LIN {X 0,Y 258.758,Z 885.566,A -85,B 0,C 180,E1 12350.11,E2 12350.11} C_VEL
LIN {X 0,Y 258.818,Z 883.349,A -85,B 0,C 180,E1 12346.376,E2 12346.376} C_VEL
LIN {X 0,Y 259.397,Z 879.488,A -85,B 0,C 180,E1 12342.915,E2 12342.915} C_VEL
LIN {X 0,Y 260.526,Z 873.775,A -85,B 0,C 180,E1 12339.483,E2 12339.483} C_VEL
LIN {X 0,Y 262.114,Z 866.611,A -85,B 0,C 180,E1 12336.348,E2 12336.348} C_VEL
LIN {X 0,Y 264.269,Z 857.295,A -85,B 0,C 180,E1 12333.25,E2 12333.25} C_VEL
LIN {X 0,Y 266.549,Z 847.181,A -85,B 0,C 180,E1 12330.642,E2 12330.642} C_VEL
LIN {X 0,Y 269.099,Z 835.15,A -85,B 0,C 180,E1 12328.192,E2 12328.192} C_VEL
LIN {X 0,Y 271.468,Z 822.672,A -85,B 0,C 180,E1 12326.196,E2 12326.196} C_VEL
LIN {X 0,Y 273.929,Z 807.744,A -85,B 0,C 180,E1 12324.342,E2 12324.342} C_VEL
LIN {X 0,Y 275.918,Z 792.384,A -85,B 0,C 180,E1 12322.921,E2 12322.921} C_VEL
LIN {X 0,Y 277.442,Z 776.257,A -85,B 0,C 180,E1 12321.847,E2 12321.847} C_VEL
LIN {X 0,Y 278.409,Z 758.677,A -85,B 0,C 180,E1 12321.115,E2 12321.115} C_VEL
LIN {X 0,Y 281.706,Z 674.031,A -85,B 0,C 180,E1 12318.89,E2 12318.89} C_VEL
LIN {X 0,Y 275.076,Z 627.916,A -85,B 0,C 180,E1 12316.6,E2 12316.6} C_VEL
LIN {X 0,Y 278.512,Z 610.893,A -85,B 0,C 180,E1 12313.201,E2 12313.201} C_VEL
LIN {X 0,Y 275.324,Z 596.958,A -85,B 0,C 180,E1 12309.373,E2 12309.373} C_VEL
LIN {X 0,Y 271.574,Z 583.053,A -85,B 0,C 180,E1 12305.183,E2 12305.183} C_VEL
LIN {X 0,Y 267.885,Z 571.432,A -85,B 0,C 180,E1 12301.298,E2 12301.298} C_VEL
LIN {X 0,Y 264.194,Z 560.871,A -85,B 0,C 180,E1 12297.38,E2 12297.38} C_VEL
LIN {X 0,Y 260.854,Z 552.791,A -85,B 0,C 180,E1 12293.977,E2 12293.977} C_VEL
LIN {X 0,Y 259.488,Z 549.45,A -85,B 0,C 180,E1 12292.497,E2 12292.497} C_VEL
LIN {X 0,Y 258.561,Z 546.696,A -85,B 0,C 180,E1 12291.159,E2 12291.159} C_VEL
LIN {X 0,Y 258.551,Z 546.561,A -85,B 0,C 180,E1 12286.317,E2 12286.317} C_VEL
LIN {X 0,Y 258.532,Z 546.552,A -85,B 0,C 180,E1 12281.386,E2 12281.386} C_VEL
LIN {X 0,Y 258.556,Z 546.573,A -85,B 0,C 180,E1 12276.551,E2 12276.551} C_VEL
LIN {X 0,Y 258.554,Z 546.567,A -85,B 0,C 180,E1 12271.708,E2 12271.708} C_VEL
LIN {X 0,Y 258.569,Z 546.551,A -85,B 0,C 180,E1 12267.961,E2 12267.961} C_VEL
LIN {X 0,Y 257.69,Z 546.65,A -85,B 0,C 180,E1 12266.375,E2 12266.375} C_VEL
LIN {X 0,Y 254.009,Z 547.136,A -85,B 0,C 180,E1 12263.744,E2 12263.744} C_VEL
LIN {X 0,Y 250.939,Z 547.534,A -85,B 0,C 180,E1 12261.149,E2 12261.149} C_VEL
LIN {X 0,Y 250.622,Z 547.549,A -85,B 0,C 180,E1 12260.125,E2 12260.125} C_VEL
LIN {X 0,Y 250.618,Z 547.547,A -85,B 0,C 180,E1 12255.107,E2 12255.107} C_VEL
LIN {X 0,Y 250.613,Z 547.525,A -85,B 0,C 180,E1 12250.111,E2 12250.111} C_VEL
LIN {X 0,Y 250.638,Z 547.568,A -85,B 0,C 180,E1 12245.265,E2 12245.265} C_VEL
LIN {X 0,Y 250.61,Z 547.52,A -85,B 0,C 180,E1 12240.229,E2 12240.229} C_VEL
LIN {X 0,Y 250.638,Z 547.563,A -85,B 0,C 180,E1 12235.195,E2 12235.195} C_VEL
LIN {X 0,Y 250.628,Z 547.546,A -85,B 0,C 180,E1 12230.355,E2 12230.355} C_VEL
LIN {X 0,Y 250.629,Z 547.535,A -85,B 0,C 180,E1 12225.208,E2 12225.208} C_VEL
LIN {X 0,Y 250.642,Z 547.549,A -85,B 0,C 180,E1 12220.29,E2 12220.29} C_VEL
LIN {X 0,Y 250.686,Z 547.86,A -85,B 0,C 180,E1 12216.759,E2 12216.759} C_VEL
LIN {X 0,Y 252.116,Z 551.307,A -85,B 0,C 180,E1 12215.142,E2 12215.142} C_VEL
LIN {X 0,Y 254.863,Z 557.484,A -85,B 0,C 180,E1 12212.449,E2 12212.449} C_VEL
LIN {X 0,Y 258.133,Z 564.923,A -85,B 0,C 180,E1 12209.508,E2 12209.508} C_VEL
LIN {X 0,Y 262.832,Z 576.542,A -85,B 0,C 180,E1 12205.471,E2 12205.471} C_VEL
LIN {X 0,Y 267.413,Z 589.235,A -85,B 0,C 180,E1 12201.635,E2 12201.635} C_VEL
LIN {X 0,Y 272.139,Z 603.788,A -85,B 0,C 180,E1 12197.751,E2 12197.751} C_VEL
LIN {X 0,Y 276.856,Z 619.87,A -85,B 0,C 180,E1 12193.999,E2 12193.999} C_VEL
LIN {X 0,Y 277.573,Z 622.236,A -85,B 0,C 180,E1 12193.816,E2 12193.816} C_VEL
LIN {X 0,Y 280.008,Z 658.39,A -85,B 0,C 180,E1 12192.396,E2 12192.396} C_VEL
LIN {X 0,Y 274.15,Z 803.54,A -85,B 0,C 180,E1 12188.817,E2 12188.817} C_VEL
LIN {X 0,Y 272.525,Z 821.816,A -85,B 0,C 180,E1 12188.018,E2 12188.018} C_VEL
LIN {X 0,Y 270.06,Z 839.883,A -85,B 0,C 180,E1 12186.854,E2 12186.854} C_VEL
LIN {X 0,Y 267.199,Z 856.691,A -85,B 0,C 180,E1 12185.367,E2 12185.367} C_VEL
LIN {X 0,Y 263.969,Z 873.171,A -85,B 0,C 180,E1 12183.457,E2 12183.457} C_VEL
LIN {X 0,Y 260.659,Z 888.442,A -85,B 0,C 180,E1 12181.188,E2 12181.188} C_VEL
LIN {X 0,Y 257.395,Z 902.672,A -85,B 0,C 180,E1 12178.542,E2 12178.542} C_VEL
LIN {X 0,Y 254.546,Z 915.418,A -85,B 0,C 180,E1 12175.6,E2 12175.6} C_VEL
LIN {X 0,Y 252.179,Z 926.751,A -85,B 0,C 180,E1 12172.374,E2 12172.374} C_VEL
LIN {X 0,Y 250.447,Z 936.689,A -85,B 0,C 180,E1 12168.868,E2 12168.868} C_VEL
LIN {X 0,Y 249.449,Z 945.396,A -85,B 0,C 180,E1 12164.986,E2 12164.986} C_VEL
LIN {X 0,Y 249.259,Z 952.053,A -85,B 0,C 180,E1 12161.103,E2 12161.103} C_VEL
LIN {X 0,Y 249.653,Z 956.774,A -85,B 0,C 180,E1 12157.365,E2 12157.365} C_VEL
LIN {X 0,Y 250.277,Z 959.854,A -85,B 0,C 180,E1 12153.667,E2 12153.667} C_VEL
LIN {X 0,Y 250.57,Z 961.172,A -85,B 0,C 180,E1 12150.46,E2 12150.46} C_VEL
LIN {X 0,Y 250.268,Z 961.223,A -85,B 0,C 180,E1 12147.175,E2 12147.175} C_VEL
LIN {X 0,Y 249.549,Z 959.846,A -85,B 0,C 180,E1 12143.539,E2 12143.539} C_VEL
LIN {X 0,Y 249.003,Z 956.775,A -85,B 0,C 180,E1 12139.594,E2 12139.594} C_VEL
LIN {X 0,Y 249.15,Z 951.57,A -85,B 0,C 180,E1 12135.273,E2 12135.273} C_VEL
LIN {X 0,Y 250.324,Z 944.676,A -85,B 0,C 180,E1 12131.128,E2 12131.128} C_VEL
LIN {X 0,Y 252.559,Z 936.103,A -85,B 0,C 180,E1 12127.177,E2 12127.177} C_VEL
LIN {X 0,Y 255.721,Z 926.051,A -85,B 0,C 180,E1 12123.535,E2 12123.535} C_VEL
LIN {X 0,Y 259.604,Z 914.488,A -85,B 0,C 180,E1 12120.215,E2 12120.215} C_VEL
LIN {X 0,Y 263.919,Z 901.943,A -85,B 0,C 180,E1 12117.332,E2 12117.332} C_VEL
LIN {X 0,Y 268.723,Z 887.471,A -85,B 0,C 180,E1 12114.688,E2 12114.688} C_VEL
LIN {X 0,Y 273.382,Z 872.233,A -85,B 0,C 180,E1 12112.493,E2 12112.493} C_VEL
LIN {X 0,Y 277.765,Z 856.171,A -85,B 0,C 180,E1 12110.696,E2 12110.696} C_VEL
LIN {X 0,Y 281.501,Z 840.182,A -85,B 0,C 180,E1 12109.332,E2 12109.332} C_VEL
LIN {X 0,Y 284.793,Z 822.514,A -85,B 0,C 180,E1 12108.235,E2 12108.235} C_VEL
LIN {X 0,Y 287.088,Z 804.522,A -85,B 0,C 180,E1 12107.461,E2 12107.461} C_VEL
LIN {X 0,Y 288.669,Z 779.142,A -85,B 0,C 180,E1 12106.785,E2 12106.785} C_VEL
LIN {X 0,Y 295.03,Z 657.964,A -85,B 0,C 180,E1 12103.843,E2 12103.843} C_VEL
LIN {X 0,Y 293.51,Z 637.024,A -85,B 0,C 180,E1 12102.746,E2 12102.746} C_VEL
LIN {X 0,Y 286.069,Z 624.221,A -85,B 0,C 180,E1 12100.516,E2 12100.516} C_VEL
LIN {X 0,Y 284.077,Z 620.553,A -85,B 0,C 180,E1 12099.769,E2 12099.769} C_VEL
LIN {X 0,Y 280.84,Z 610.811,A -85,B 0,C 180,E1 12096.228,E2 12096.228} C_VEL
LIN {X 0,Y 277.656,Z 602.086,A -85,B 0,C 180,E1 12092.449,E2 12092.449} C_VEL
LIN {X 0,Y 274.616,Z 594.628,A -85,B 0,C 180,E1 12088.487,E2 12088.487} C_VEL
LIN {X 0,Y 272.578,Z 590.196,A -85,B 0,C 180,E1 12085.546,E2 12085.546} C_VEL
LIN {X 0,Y 271.016,Z 586.561,A -85,B 0,C 180,E1 12082.791,E2 12082.791} C_VEL
LIN {X 0,Y 269.161,Z 582.502,A -85,B 0,C 180,E1 12078.855,E2 12078.855} C_VEL
LIN {X 0,Y 267.28,Z 578.403,A -85,B 0,C 180,E1 12072.311,E2 12072.311} C_VEL
LIN {X 0,Y 266.55,Z 577.578,A -85,B 0,C 180,E1 12067.11,E2 12067.11} C_VEL
LIN {X 0,Y 266.942,Z 578.179,A -85,B 0,C 180,E1 12062.146,E2 12062.146} C_VEL
LIN {X 0,Y 268.477,Z 582.356,A -85,B 0,C 180,E1 12055.086,E2 12055.086} C_VEL
LIN {X 0,Y 269.944,Z 586.327,A -85,B 0,C 180,E1 12051.05,E2 12051.05} C_VEL
LIN {X 0,Y 271.377,Z 590.311,A -85,B 0,C 180,E1 12047.877,E2 12047.877} C_VEL
LIN {X 0,Y 273.341,Z 595.613,A -85,B 0,C 180,E1 12044.294,E2 12044.294} C_VEL
LIN {X 0,Y 275.612,Z 602.962,A -85,B 0,C 180,E1 12040.282,E2 12040.282} C_VEL
LIN {X 0,Y 277.948,Z 611.166,A -85,B 0,C 180,E1 12036.465,E2 12036.465} C_VEL
LIN {X 0,Y 280.209,Z 620.765,A -85,B 0,C 180,E1 12032.67,E2 12032.67} C_VEL
LIN {X 0,Y 281.533,Z 627.351,A -85,B 0,C 180,E1 12030.418,E2 12030.418} C_VEL
LIN {X 0,Y 283.668,Z 632.135,A -85,B 0,C 180,E1 12029.615,E2 12029.615} C_VEL
LIN {X 0,Y 288.538,Z 660.508,A -85,B 0,C 180,E1 12027.323,E2 12027.323} C_VEL
LIN {X 0,Y 291.484,Z 682.296,A -85,B 0,C 180,E1 12025.844,E2 12025.844} C_VEL
LIN {X 0,Y 286.431,Z 766.945,A -85,B 0,C 180,E1 12023.607,E2 12023.607} C_VEL
LIN {X 0,Y 284.87,Z 783.092,A -85,B 0,C 180,E1 12022.841,E2 12022.841} C_VEL
LIN {X 0,Y 282.515,Z 798.96,A -85,B 0,C 180,E1 12021.731,E2 12021.731} C_VEL
LIN {X 0,Y 279.664,Z 813.068,A -85,B 0,C 180,E1 12020.385,E2 12020.385} C_VEL
LIN {X 0,Y 276.006,Z 827.571,A -85,B 0,C 180,E1 12018.57,E2 12018.57} C_VEL
LIN {X 0,Y 272.149,Z 840.225,A -85,B 0,C 180,E1 12016.51,E2 12016.51} C_VEL
LIN {X 0,Y 268.136,Z 851.743,A -85,B 0,C 180,E1 12014.096,E2 12014.096} C_VEL
LIN {X 0,Y 264.287,Z 861.551,A -85,B 0,C 180,E1 12011.45,E2 12011.45} C_VEL
LIN {X 0,Y 260.567,Z 870.116,A -85,B 0,C 180,E1 12008.428,E2 12008.428} C_VEL
LIN {X 0,Y 257.479,Z 876.685,A -85,B 0,C 180,E1 12005.346,E2 12005.346} C_VEL
LIN {X 0,Y 254.698,Z 882.07,A -85,B 0,C 180,E1 12001.732,E2 12001.732} C_VEL
LIN {X 0,Y 252.737,Z 885.492,A -85,B 0,C 180,E1 11998.079,E2 11998.079} C_VEL
LIN {X 0,Y 251.438,Z 887.087,A -85,B 0,C 180,E1 11994.174,E2 11994.174} C_VEL
LIN {X 0,Y 250.871,Z 886.852,A -85,B 0,C 180,E1 11990.509,E2 11990.509} C_VEL
LIN {X 0,Y 250.867,Z 884.74,A -85,B 0,C 180,E1 11986.672,E2 11986.672} C_VEL
LIN {X 0,Y 251.439,Z 880.947,A -85,B 0,C 180,E1 11983.027,E2 11983.027} C_VEL
LIN {X 0,Y 252.635,Z 875.05,A -85,B 0,C 180,E1 11979.335,E2 11979.335} C_VEL
LIN {X 0,Y 254.287,Z 867.913,A -85,B 0,C 180,E1 11976.091,E2 11976.091} C_VEL
LIN {X 0,Y 256.52,Z 858.641,A -85,B 0,C 180,E1 11972.901,E2 11972.901} C_VEL
LIN {X 0,Y 258.967,Z 848.269,A -85,B 0,C 180,E1 11970.137,E2 11970.137} C_VEL
LIN {X 0,Y 261.661,Z 836.084,A -85,B 0,C 180,E1 11967.589,E2 11967.589} C_VEL
LIN {X 0,Y 264.264,Z 822.893,A -85,B 0,C 180,E1 11965.441,E2 11965.441} C_VEL
LIN {X 0,Y 266.674,Z 808.828,A -85,B 0,C 180,E1 11963.658,E2 11963.658} C_VEL
LIN {X 0,Y 268.614,Z 794.73,A -85,B 0,C 180,E1 11962.297,E2 11962.297} C_VEL
LIN {X 0,Y 270.317,Z 777.953,A -85,B 0,C 180,E1 11961.121,E2 11961.121} C_VEL
LIN {X 0,Y 271.331,Z 761.274,A -85,B 0,C 180,E1 11960.379,E2 11960.379} C_VEL
LIN {X 0,Y 274.846,Z 675.092,A -85,B 0,C 180,E1 11958.055,E2 11958.055} C_VEL
LIN {X 0,Y 268.186,Z 627.499,A -85,B 0,C 180,E1 11955.589,E2 11955.589} C_VEL
LIN {X 0,Y 271.201,Z 613.467,A -85,B 0,C 180,E1 11952.724,E2 11952.724} C_VEL
LIN {X 0,Y 268.053,Z 599.58,A -85,B 0,C 180,E1 11948.787,E2 11948.787} C_VEL
LIN {X 0,Y 264.589,Z 586.434,A -85,B 0,C 180,E1 11944.721,E2 11944.721} C_VEL
LIN {X 0,Y 260.789,Z 574.229,A -85,B 0,C 180,E1 11940.496,E2 11940.496} C_VEL
LIN {X 0,Y 257.249,Z 564.413,A -85,B 0,C 180,E1 11936.684,E2 11936.684} C_VEL
LIN {X 0,Y 253.65,Z 555.043,A -85,B 0,C 180,E1 11932.624,E2 11932.624} C_VEL
LIN {X 0,Y 251.624,Z 550.587,A -85,B 0,C 180,E1 11930.434,E2 11930.434} C_VEL
LIN {X 0,Y 250.629,Z 547.642,A -85,B 0,C 180,E1 11928.834,E2 11928.834} C_VEL
LIN {X 0,Y 250.605,Z 547.576,A -85,B 0,C 180,E1 11923.966,E2 11923.966} C_VEL
LIN {X 0,Y 250.612,Z 547.562,A -85,B 0,C 180,E1 11918.784,E2 11918.784} C_VEL
LIN {X 0,Y 250.614,Z 547.529,A -85,B 0,C 180,E1 11913.92,E2 11913.92} C_VEL
LIN {X 0,Y 250.605,Z 547.561,A -85,B 0,C 180,E1 11908.867,E2 11908.867} C_VEL
LIN {X 0,Y 250.63,Z 547.541,A -85,B 0,C 180,E1 11904.001,E2 11904.001} C_VEL
LIN {X 0,Y 250.622,Z 547.549,A -85,B 0,C 180,E1 11900.125,E2 11900.125} C_VEL
LIN {X 0,Y 249.791,Z 547.637,A -85,B 0,C 180,E1 11898.488,E2 11898.488} C_VEL
LIN {X 0,Y 246.304,Z 548.106,A -85,B 0,C 180,E1 11895.898,E2 11895.898} C_VEL
LIN {X 0,Y 243.012,Z 548.531,A -85,B 0,C 180,E1 11893.093,E2 11893.093} C_VEL
LIN {X 0,Y 242.68,Z 548.551,A -85,B 0,C 180,E1 11892.034,E2 11892.034} C_VEL
LIN {X 0,Y 242.69,Z 548.515,A -85,B 0,C 180,E1 11887.1,E2 11887.1} C_VEL
LIN {X 0,Y 242.673,Z 548.522,A -85,B 0,C 180,E1 11882.126,E2 11882.126} C_VEL
LIN {X 0,Y 242.696,Z 548.552,A -85,B 0,C 180,E1 11877.167,E2 11877.167} C_VEL
LIN {X 0,Y 242.68,Z 548.516,A -85,B 0,C 180,E1 11872.186,E2 11872.186} C_VEL
LIN {X 0,Y 242.695,Z 548.54,A -85,B 0,C 180,E1 11867.146,E2 11867.146} C_VEL
LIN {X 0,Y 242.701,Z 548.561,A -85,B 0,C 180,E1 11862.251,E2 11862.251} C_VEL
LIN {X 0,Y 242.737,Z 548.869,A -85,B 0,C 180,E1 11859.312,E2 11859.312} C_VEL
LIN {X 0,Y 244.971,Z 553.954,A -85,B 0,C 180,E1 11856.678,E2 11856.678} C_VEL
LIN {X 0,Y 247.097,Z 558.693,A -85,B 0,C 180,E1 11854.465,E2 11854.465} C_VEL
LIN {X 0,Y 250.127,Z 565.32,A -85,B 0,C 180,E1 11851.57,E2 11851.57} C_VEL
LIN {X 0,Y 254.559,Z 576.319,A -85,B 0,C 180,E1 11847.445,E2 11847.445} C_VEL
LIN {X 0,Y 259.008,Z 588.256,A -85,B 0,C 180,E1 11843.524,E2 11843.524} C_VEL
LIN {X 0,Y 263.755,Z 602.506,A -85,B 0,C 180,E1 11839.449,E2 11839.449} C_VEL
LIN {X 0,Y 268.597,Z 619.006,A -85,B 0,C 180,E1 11835.287,E2 11835.287} C_VEL
LIN {X 0,Y 269.789,Z 621.934,A -85,B 0,C 180,E1 11834.902,E2 11834.902} C_VEL
LIN {X 0,Y 270.98,Z 624.901,A -85,B 0,C 180,E1 11834.639,E2 11834.639} C_VEL
LIN {X 0,Y 273.194,Z 659.153,A -85,B 0,C 180,E1 11833.257,E2 11833.257} C_VEL
LIN {X 0,Y 267.15,Z 803.024,A -85,B 0,C 180,E1 11829.643,E2 11829.643} C_VEL
LIN {X 0,Y 265.475,Z 821.264,A -85,B 0,C 180,E1 11828.826,E2 11828.826} C_VEL
LIN {X 0,Y 262.989,Z 838.888,A -85,B 0,C 180,E1 11827.67,E2 11827.67} C_VEL
LIN {X 0,Y 260.021,Z 855.79,A -85,B 0,C 180,E1 11826.147,E2 11826.147} C_VEL
LIN {X 0,Y 256.755,Z 871.864,A -85,B 0,C 180,E1 11824.251,E2 11824.251} C_VEL
LIN {X 0,Y 253.317,Z 887.181,A -85,B 0,C 180,E1 11821.932,E2 11821.932} C_VEL
LIN {X 0,Y 249.896,Z 901.455,A -85,B 0,C 180,E1 11819.218,E2 11819.218} C_VEL
LIN {X 0,Y 246.907,Z 914.234,A -85,B 0,C 180,E1 11816.194,E2 11816.194} C_VEL
LIN {X 0,Y 244.415,Z 925.589,A -85,B 0,C 180,E1 11812.87,E2 11812.87} C_VEL
LIN {X 0,Y 242.579,Z 935.542,A -85,B 0,C 180,E1 11809.254,E2 11809.254} C_VEL
LIN {X 0,Y 241.522,Z 944.164,A -85,B 0,C 180,E1 11805.296,E2 11805.296} C_VEL
LIN {X 0,Y 241.3,Z 950.922,A -85,B 0,C 180,E1 11801.232,E2 11801.232} C_VEL
LIN {X 0,Y 241.715,Z 955.639,A -85,B 0,C 180,E1 11797.37,E2 11797.37} C_VEL
LIN {X 0,Y 242.377,Z 958.702,A -85,B 0,C 180,E1 11793.55,E2 11793.55} C_VEL
LIN {X 0,Y 242.665,Z 959.998,A -85,B 0,C 180,E1 11790.239,E2 11790.239} C_VEL
LIN {X 0,Y 242.3,Z 960.012,A -85,B 0,C 180,E1 11786.928,E2 11786.928} C_VEL
LIN {X 0,Y 241.518,Z 958.58,A -85,B 0,C 180,E1 11783.108,E2 11783.108} C_VEL
LIN {X 0,Y 240.994,Z 955.442,A -85,B 0,C 180,E1 11779.002,E2 11779.002} C_VEL
LIN {X 0,Y 241.266,Z 950.307,A -85,B 0,C 180,E1 11774.624,E2 11774.624} C_VEL
LIN {X 0,Y 242.667,Z 943.23,A -85,B 0,C 180,E1 11770.258,E2 11770.258} C_VEL
LIN {X 0,Y 245.175,Z 934.596,A -85,B 0,C 180,E1 11766.193,E2 11766.193} C_VEL
LIN {X 0,Y 248.639,Z 924.487,A -85,B 0,C 180,E1 11762.46,E2 11762.46} C_VEL
LIN {X 0,Y 252.834,Z 912.848,A -85,B 0,C 180,E1 11759.069,E2 11759.069} C_VEL
LIN {X 0,Y 257.636,Z 899.678,A -85,B 0,C 180,E1 11756.03,E2 11756.03} C_VEL
LIN {X 0,Y 262.463,Z 885.824,A -85,B 0,C 180,E1 11753.495,E2 11753.495} C_VEL
LIN {X 0,Y 267.231,Z 870.909,A -85,B 0,C 180,E1 11751.337,E2 11751.337} C_VEL
LIN {X 0,Y 271.819,Z 854.755,A -85,B 0,C 180,E1 11749.524,E2 11749.524} C_VEL
LIN {X 0,Y 275.862,Z 837.898,A -85,B 0,C 180,E1 11748.108,E2 11748.108} C_VEL
LIN {X 0,Y 279.204,Z 820.161,A -85,B 0,C 180,E1 11747.027,E2 11747.027} C_VEL
LIN {X 0,Y 281.553,Z 801.605,A -85,B 0,C 180,E1 11746.251,E2 11746.251} C_VEL
LIN {X 0,Y 283.744,Z 764.34,A -85,B 0,C 180,E1 11745.305,E2 11745.305} C_VEL
LIN {X 0,Y 289.594,Z 658.934,A -85,B 0,C 180,E1 11742.7,E2 11742.7} C_VEL
LIN {X 0,Y 288.373,Z 641.068,A -85,B 0,C 180,E1 11741.736,E2 11741.736} C_VEL
LIN {X 0,Y 280.607,Z 627.479,A -85,B 0,C 180,E1 11739.265,E2 11739.265} C_VEL
LIN {X 0,Y 276.601,Z 620.847,A -85,B 0,C 180,E1 11737.753,E2 11737.753} C_VEL
LIN {X 0,Y 273.257,Z 611.063,A -85,B 0,C 180,E1 11733.791,E2 11733.791} C_VEL
LIN {X 0,Y 270.295,Z 603.354,A -85,B 0,C 180,E1 11729.959,E2 11729.959} C_VEL
LIN {X 0,Y 267.793,Z 597.058,A -85,B 0,C 180,E1 11726.14,E2 11726.14} C_VEL
LIN {X 0,Y 265.692,Z 592.469,A -85,B 0,C 180,E1 11722.572,E2 11722.572} C_VEL
LIN {X 0,Y 264.006,Z 588.611,A -85,B 0,C 180,E1 11718.779,E2 11718.779} C_VEL
LIN {X 0,Y 262.172,Z 584.562,A -85,B 0,C 180,E1 11712.331,E2 11712.331} C_VEL
LIN {X 0,Y 261.41,Z 583.713,A -85,B 0,C 180,E1 11707.03,E2 11707.03} C_VEL
LIN {X 0,Y 261.77,Z 584.358,A -85,B 0,C 180,E1 11701.97,E2 11701.97} C_VEL
LIN {X 0,Y 263.12,Z 588.296,A -85,B 0,C 180,E1 11695.204,E2 11695.204} C_VEL
LIN {X 0,Y 264.525,Z 592.307,A -85,B 0,C 180,E1 11691.084,E2 11691.084} C_VEL
LIN {X 0,Y 265.874,Z 596.287,A -85,B 0,C 180,E1 11687.842,E2 11687.842} C_VEL
LIN {X 0,Y 267.657,Z 601.313,A -85,B 0,C 180,E1 11684.397,E2 11684.397} C_VEL
LIN {X 0,Y 269.971,Z 609.092,A -85,B 0,C 180,E1 11680.078,E2 11680.078} C_VEL
LIN {X 0,Y 272.166,Z 617.547,A -85,B 0,C 180,E1 11676.153,E2 11676.153} C_VEL
LIN {X 0,Y 274.175,Z 626.767,A -85,B 0,C 180,E1 11672.527,E2 11672.527} C_VEL
LIN {X 0,Y 278.927,Z 636.071,A -85,B 0,C 180,E1 11670.675,E2 11670.675} C_VEL
LIN {X 0,Y 283.381,Z 663.273,A -85,B 0,C 180,E1 11668.416,E2 11668.416} C_VEL
LIN {X 0,Y 286.018,Z 683.721,A -85,B 0,C 180,E1 11666.987,E2 11666.987} C_VEL
LIN {X 0,Y 280.793,Z 767.637,A -85,B 0,C 180,E1 11664.746,E2 11664.746} C_VEL
LIN {X 0,Y 279.152,Z 783.83,A -85,B 0,C 180,E1 11663.969,E2 11663.969} C_VEL
LIN {X 0,Y 276.671,Z 799.801,A -85,B 0,C 180,E1 11662.838,E2 11662.838} C_VEL
LIN {X 0,Y 273.599,Z 814.23,A -85,B 0,C 180,E1 11661.439,E2 11661.439} C_VEL
LIN {X 0,Y 269.746,Z 828.724,A -85,B 0,C 180,E1 11659.59,E2 11659.59} C_VEL
LIN {X 0,Y 265.72,Z 841.244,A -85,B 0,C 180,E1 11657.511,E2 11657.511} C_VEL
LIN {X 0,Y 261.301,Z 853.247,A -85,B 0,C 180,E1 11654.935,E2 11654.935} C_VEL
LIN {X 0,Y 257.266,Z 862.926,A -85,B 0,C 180,E1 11652.241,E2 11652.241} C_VEL
LIN {X 0,Y 253.347,Z 871.438,A -85,B 0,C 180,E1 11649.15,E2 11649.15} C_VEL
LIN {X 0,Y 250.075,Z 877.958,A -85,B 0,C 180,E1 11645.99,E2 11645.99} C_VEL
LIN {X 0,Y 247.096,Z 883.341,A -85,B 0,C 180,E1 11642.251,E2 11642.251} C_VEL
LIN {X 0,Y 245.006,Z 886.709,A -85,B 0,C 180,E1 11638.514,E2 11638.514} C_VEL
LIN {X 0,Y 243.597,Z 888.292,A -85,B 0,C 180,E1 11634.486,E2 11634.486} C_VEL
LIN {X 0,Y 242.971,Z 888.056,A -85,B 0,C 180,E1 11630.721,E2 11630.721} C_VEL
LIN {X 0,Y 242.938,Z 885.938,A -85,B 0,C 180,E1 11626.74,E2 11626.74} C_VEL
LIN {X 0,Y 243.5,Z 882.258,A -85,B 0,C 180,E1 11623.048,E2 11623.048} C_VEL
LIN {X 0,Y 244.651,Z 876.713,A -85,B 0,C 180,E1 11619.405,E2 11619.405} C_VEL
LIN {X 0,Y 246.333,Z 869.723,A -85,B 0,C 180,E1 11616.034,E2 11616.034} C_VEL
LIN {X 0,Y 248.591,Z 860.689,A -85,B 0,C 180,E1 11612.763,E2 11612.763} C_VEL
LIN {X 0,Y 251.015,Z 850.942,A -85,B 0,C 180,E1 11609.997,E2 11609.997} C_VEL
LIN {X 0,Y 253.732,Z 839.277,A -85,B 0,C 180,E1 11607.4,E2 11607.4} C_VEL
LIN {X 0,Y 256.535,Z 826.024,A -85,B 0,C 180,E1 11605.079,E2 11605.079} C_VEL
LIN {X 0,Y 259.178,Z 811.47,A -85,B 0,C 180,E1 11603.129,E2 11603.129} C_VEL
LIN {X 0,Y 261.336,Z 796.944,A -85,B 0,C 180,E1 11601.638,E2 11601.638} C_VEL
LIN {X 0,Y 263.132,Z 780.437,A -85,B 0,C 180,E1 11600.421,E2 11600.421} C_VEL
LIN {X 0,Y 264.262,Z 764.216,A -85,B 0,C 180,E1 11599.628,E2 11599.628} C_VEL
LIN {X 0,Y 267.998,Z 676.088,A -85,B 0,C 180,E1 11597.186,E2 11597.186} C_VEL
LIN {X 0,Y 261.343,Z 627.714,A -85,B 0,C 180,E1 11594.606,E2 11594.606} C_VEL
LIN {X 0,Y 263.831,Z 615.702,A -85,B 0,C 180,E1 11592.122,E2 11592.122} C_VEL
LIN {X 0,Y 260.776,Z 601.953,A -85,B 0,C 180,E1 11588.106,E2 11588.106} C_VEL
LIN {X 0,Y 257.4,Z 589.044,A -85,B 0,C 180,E1 11583.963,E2 11583.963} C_VEL
LIN {X 0,Y 253.675,Z 577.144,A -85,B 0,C 180,E1 11579.677,E2 11579.677} C_VEL
LIN {X 0,Y 250.192,Z 567.11,A -85,B 0,C 180,E1 11575.635,E2 11575.635} C_VEL
LIN {X 0,Y 246.799,Z 558.83,A -85,B 0,C 180,E1 11571.81,E2 11571.81} C_VEL
LIN {X 0,Y 245.287,Z 555.284,A -85,B 0,C 180,E1 11570.027,E2 11570.027} C_VEL
LIN {X 0,Y 243.895,Z 551.902,A -85,B 0,C 180,E1 11568.256,E2 11568.256} C_VEL
LIN {X 0,Y 242.694,Z 548.684,A -85,B 0,C 180,E1 11566.381,E2 11566.381} C_VEL
LIN {X 0,Y 242.655,Z 548.527,A -85,B 0,C 180,E1 11561.246,E2 11561.246} C_VEL
LIN {X 0,Y 242.682,Z 548.543,A -85,B 0,C 180,E1 11556.391,E2 11556.391} C_VEL
LIN {X 0,Y 242.667,Z 548.552,A -85,B 0,C 180,E1 11551.276,E2 11551.276} C_VEL
LIN {X 0,Y 242.683,Z 548.509,A -85,B 0,C 180,E1 11546.158,E2 11546.158} C_VEL
LIN {X 0,Y 242.679,Z 548.564,A -85,B 0,C 180,E1 11541.259,E2 11541.259} C_VEL
LIN {X 0,Y 242.68,Z 548.516,A -85,B 0,C 180,E1 11536.025,E2 11536.025} C_VEL
LIN {X 0,Y 242.68,Z 548.551,A -85,B 0,C 180,E1 11532.034,E2 11532.034} C_VEL
LIN {X 0,Y 241.836,Z 548.633,A -85,B 0,C 180,E1 11530.344,E2 11530.344} C_VEL
LIN {X 0,Y 238.349,Z 549.094,A -85,B 0,C 180,E1 11527.667,E2 11527.667} C_VEL
LIN {X 0,Y 235.072,Z 549.519,A -85,B 0,C 180,E1 11524.766,E2 11524.766} C_VEL
LIN {X 0,Y 234.747,Z 549.542,A -85,B 0,C 180,E1 11523.672,E2 11523.672} C_VEL
LIN {X 0,Y 234.751,Z 549.505,A -85,B 0,C 180,E1 11518.78,E2 11518.78} C_VEL
LIN {X 0,Y 234.742,Z 549.511,A -85,B 0,C 180,E1 11513.642,E2 11513.642} C_VEL
LIN {X 0,Y 234.765,Z 549.556,A -85,B 0,C 180,E1 11508.702,E2 11508.702} C_VEL
LIN {X 0,Y 234.748,Z 549.525,A -85,B 0,C 180,E1 11503.397,E2 11503.397} C_VEL
LIN {X 0,Y 234.813,Z 549.902,A -85,B 0,C 180,E1 11502.211,E2 11502.211} C_VEL
LIN {X 0,Y 236.511,Z 553.639,A -85,B 0,C 180,E1 11499.975,E2 11499.975} C_VEL
LIN {X 0,Y 239.177,Z 559.522,A -85,B 0,C 180,E1 11496.862,E2 11496.862} C_VEL
LIN {X 0,Y 242.464,Z 566.618,A -85,B 0,C 180,E1 11493.486,E2 11493.486} C_VEL
LIN {X 0,Y 246.915,Z 577.538,A -85,B 0,C 180,E1 11489.051,E2 11489.051} C_VEL
LIN {X 0,Y 251.237,Z 588.998,A -85,B 0,C 180,E1 11485.035,E2 11485.035} C_VEL
LIN {X 0,Y 255.941,Z 603.128,A -85,B 0,C 180,E1 11480.738,E2 11480.738} C_VEL
LIN {X 0,Y 260.38,Z 618.15,A -85,B 0,C 180,E1 11476.73,E2 11476.73} C_VEL
LIN {X 0,Y 261.29,Z 620.86,A -85,B 0,C 180,E1 11476.201,E2 11476.201} C_VEL
LIN {X 0,Y 264.444,Z 627.738,A -85,B 0,C 180,E1 11475.492,E2 11475.492} C_VEL
LIN {X 0,Y 266.429,Z 659.847,A -85,B 0,C 180,E1 11474.159,E2 11474.159} C_VEL
LIN {X 0,Y 260.175,Z 802.403,A -85,B 0,C 180,E1 11470.501,E2 11470.501} C_VEL
LIN {X 0,Y 258.451,Z 820.641,A -85,B 0,C 180,E1 11469.667,E2 11469.667} C_VEL
LIN {X 0,Y 255.879,Z 838.284,A -85,B 0,C 180,E1 11468.485,E2 11468.485} C_VEL
LIN {X 0,Y 252.847,Z 855.007,A -85,B 0,C 180,E1 11466.946,E2 11466.946} C_VEL
LIN {X 0,Y 249.413,Z 871.298,A -85,B 0,C 180,E1 11464.978,E2 11464.978} C_VEL
LIN {X 0,Y 245.858,Z 886.538,A -85,B 0,C 180,E1 11462.606,E2 11462.606} C_VEL
LIN {X 0,Y 242.292,Z 900.804,A -85,B 0,C 180,E1 11459.812,E2 11459.812} C_VEL
LIN {X 0,Y 239.082,Z 913.947,A -85,B 0,C 180,E1 11456.583,E2 11456.583} C_VEL
LIN {X 0,Y 236.51,Z 925.175,A -85,B 0,C 180,E1 11453.152,E2 11453.152} C_VEL
LIN {X 0,Y 234.623,Z 935.007,A -85,B 0,C 180,E1 11449.416,E2 11449.416} C_VEL
LIN {X 0,Y 233.562,Z 943.343,A -85,B 0,C 180,E1 11445.393,E2 11445.393} C_VEL
LIN {X 0,Y 233.354,Z 950.116,A -85,B 0,C 180,E1 11441.119,E2 11441.119} C_VEL
LIN {X 0,Y 233.817,Z 954.722,A -85,B 0,C 180,E1 11437.126,E2 11437.126} C_VEL
LIN {X 0,Y 234.518,Z 957.664,A -85,B 0,C 180,E1 11433.18,E2 11433.18} C_VEL
LIN {X 0,Y 234.745,Z 958.874,A -85,B 0,C 180,E1 11429.759,E2 11429.759} C_VEL
LIN {X 0,Y 234.258,Z 958.735,A -85,B 0,C 180,E1 11426.333,E2 11426.333} C_VEL
LIN {X 0,Y 233.392,Z 957.002,A -85,B 0,C 180,E1 11422.124,E2 11422.124} C_VEL
LIN {X 0,Y 232.991,Z 953.372,A -85,B 0,C 180,E1 11417.614,E2 11417.614} C_VEL
LIN {X 0,Y 233.612,Z 947.891,A -85,B 0,C 180,E1 11413.084,E2 11413.084} C_VEL
LIN {X 0,Y 235.47,Z 940.434,A -85,B 0,C 180,E1 11408.587,E2 11408.587} C_VEL
LIN {X 0,Y 238.497,Z 931.353,A -85,B 0,C 180,E1 11404.423,E2 11404.423} C_VEL
LIN {X 0,Y 242.479,Z 920.741,A -85,B 0,C 180,E1 11400.62,E2 11400.62} C_VEL
LIN {X 0,Y 247.197,Z 908.587,A -85,B 0,C 180,E1 11397.187,E2 11397.187} C_VEL
LIN {X 0,Y 252.318,Z 895.326,A -85,B 0,C 180,E1 11394.24,E2 11394.24} C_VEL
LIN {X 0,Y 257.445,Z 880.96,A -85,B 0,C 180,E1 11391.731,E2 11391.731} C_VEL
LIN {X 0,Y 262.426,Z 865.653,A -85,B 0,C 180,E1 11389.639,E2 11389.639} C_VEL
LIN {X 0,Y 267.068,Z 849.369,A -85,B 0,C 180,E1 11387.93,E2 11387.93} C_VEL
LIN {X 0,Y 271.101,Z 832.39,A -85,B 0,C 180,E1 11386.599,E2 11386.599} C_VEL
LIN {X 0,Y 274.344,Z 814.44,A -85,B 0,C 180,E1 11385.592,E2 11385.592} C_VEL
LIN {X 0,Y 276.379,Z 796.193,A -85,B 0,C 180,E1 11384.914,E2 11384.914} C_VEL
LIN {X 0,Y 284.285,Z 660.052,A -85,B 0,C 180,E1 11381.52,E2 11381.52} C_VEL
LIN {X 0,Y 283.321,Z 645.072,A -85,B 0,C 180,E1 11380.685,E2 11380.685} C_VEL
LIN {X 0,Y 276.399,Z 632.744,A -85,B 0,C 180,E1 11378.344,E2 11378.344} C_VEL
LIN {X 0,Y 269.173,Z 621.266,A -85,B 0,C 180,E1 11375.544,E2 11375.544} C_VEL
LIN {X 0,Y 266.214,Z 612.784,A -85,B 0,C 180,E1 11371.723,E2 11371.723} C_VEL
LIN {X 0,Y 263.514,Z 605.816,A -85,B 0,C 180,E1 11367.82,E2 11367.82} C_VEL
LIN {X 0,Y 261.513,Z 601.238,A -85,B 0,C 180,E1 11364.629,E2 11364.629} C_VEL
LIN {X 0,Y 260.378,Z 598.381,A -85,B 0,C 180,E1 11362.343,E2 11362.343} C_VEL
LIN {X 0,Y 258.835,Z 594.706,A -85,B 0,C 180,E1 11358.7,E2 11358.7} C_VEL
LIN {X 0,Y 257.012,Z 590.659,A -85,B 0,C 180,E1 11352.126,E2 11352.126} C_VEL
LIN {X 0,Y 256.291,Z 589.864,A -85,B 0,C 180,E1 11346.946,E2 11346.946} C_VEL
LIN {X 0,Y 256.608,Z 590.483,A -85,B 0,C 180,E1 11342.009,E2 11342.009} C_VEL
LIN {X 0,Y 257.808,Z 594.323,A -85,B 0,C 180,E1 11335.269,E2 11335.269} C_VEL
LIN {X 0,Y 259.03,Z 598.001,A -85,B 0,C 180,E1 11331.341,E2 11331.341} C_VEL
LIN {X 0,Y 260.3,Z 601.971,A -85,B 0,C 180,E1 11328.028,E2 11328.028} C_VEL
LIN {X 0,Y 261.963,Z 607.026,A -85,B 0,C 180,E1 11324.503,E2 11324.503} C_VEL
LIN {X 0,Y 264.07,Z 614.397,A -85,B 0,C 180,E1 11320.306,E2 11320.306} C_VEL
LIN {X 0,Y 266.141,Z 622.874,A -85,B 0,C 180,E1 11316.297,E2 11316.297} C_VEL
LIN {X 0,Y 267.043,Z 626.745,A -85,B 0,C 180,E1 11314.732,E2 11314.732} C_VEL
LIN {X 0,Y 273.518,Z 638.658,A -85,B 0,C 180,E1 11312.071,E2 11312.071} C_VEL
LIN {X 0,Y 274.606,Z 641.493,A -85,B 0,C 180,E1 11311.63,E2 11311.63} C_VEL
LIN {X 0,Y 278.917,Z 670.354,A -85,B 0,C 180,E1 11309.22,E2 11309.22} C_VEL
LIN {X 0,Y 280.644,Z 685.535,A -85,B 0,C 180,E1 11308.164,E2 11308.164} C_VEL
LIN {X 0,Y 275.263,Z 768.44,A -85,B 0,C 180,E1 11305.926,E2 11305.926} C_VEL
LIN {X 0,Y 273.516,Z 784.785,A -85,B 0,C 180,E1 11305.129,E2 11305.129} C_VEL
LIN {X 0,Y 270.955,Z 800.527,A -85,B 0,C 180,E1 11304.002,E2 11304.002} C_VEL
LIN {X 0,Y 267.633,Z 815.416,A -85,B 0,C 180,E1 11302.539,E2 11302.539} C_VEL
LIN {X 0,Y 263.627,Z 829.776,A -85,B 0,C 180,E1 11300.678,E2 11300.678} C_VEL
LIN {X 0,Y 259.439,Z 842.188,A -85,B 0,C 180,E1 11298.586,E2 11298.586} C_VEL
LIN {X 0,Y 254.868,Z 853.983,A -85,B 0,C 180,E1 11296.021,E2 11296.021} C_VEL
LIN {X 0,Y 250.652,Z 863.613,A -85,B 0,C 180,E1 11293.315,E2 11293.315} C_VEL
LIN {X 0,Y 246.465,Z 872.186,A -85,B 0,C 180,E1 11290.16,E2 11290.16} C_VEL
LIN {X 0,Y 242.706,Z 879.228,A -85,B 0,C 180,E1 11286.673,E2 11286.673} C_VEL
LIN {X 0,Y 239.552,Z 884.553,A -85,B 0,C 180,E1 11282.854,E2 11282.854} C_VEL
LIN {X 0,Y 237.292,Z 887.927,A -85,B 0,C 180,E1 11278.978,E2 11278.978} C_VEL
LIN {X 0,Y 235.764,Z 889.496,A -85,B 0,C 180,E1 11274.82,E2 11274.82} C_VEL
LIN {X 0,Y 235.071,Z 889.254,A -85,B 0,C 180,E1 11270.929,E2 11270.929} C_VEL
LIN {X 0,Y 235.008,Z 887.13,A -85,B 0,C 180,E1 11266.806,E2 11266.806} C_VEL
LIN {X 0,Y 235.576,Z 883.463,A -85,B 0,C 180,E1 11262.996,E2 11262.996} C_VEL
LIN {X 0,Y 236.763,Z 877.935,A -85,B 0,C 180,E1 11259.231,E2 11259.231} C_VEL
LIN {X 0,Y 238.491,Z 871.016,A -85,B 0,C 180,E1 11255.771,E2 11255.771} C_VEL
LIN {X 0,Y 240.662,Z 862.714,A -85,B 0,C 180,E1 11252.616,E2 11252.616} C_VEL
LIN {X 0,Y 243.367,Z 852.284,A -85,B 0,C 180,E1 11249.526,E2 11249.526} C_VEL
LIN {X 0,Y 246.191,Z 840.726,A -85,B 0,C 180,E1 11246.854,E2 11246.854} C_VEL
LIN {X 0,Y 249.142,Z 827.372,A -85,B 0,C 180,E1 11244.436,E2 11244.436} C_VEL
LIN {X 0,Y 251.844,Z 813.244,A -85,B 0,C 180,E1 11242.47,E2 11242.47} C_VEL
LIN {X 0,Y 254.249,Z 797.828,A -85,B 0,C 180,E1 11240.834,E2 11240.834} C_VEL
LIN {X 0,Y 256.123,Z 781.395,A -85,B 0,C 180,E1 11239.589,E2 11239.589} C_VEL
LIN {X 0,Y 257.33,Z 764.93,A -85,B 0,C 180,E1 11238.76,E2 11238.76} C_VEL
LIN {X 0,Y 261.224,Z 677.185,A -85,B 0,C 180,E1 11236.279,E2 11236.279} C_VEL
LIN {X 0,Y 254.565,Z 627.292,A -85,B 0,C 180,E1 11233.513,E2 11233.513} C_VEL
LIN {X 0,Y 256.559,Z 618.329,A -85,B 0,C 180,E1 11231.597,E2 11231.597} C_VEL
LIN {X 0,Y 253.497,Z 604.271,A -85,B 0,C 180,E1 11227.364,E2 11227.364} C_VEL
LIN {X 0,Y 250.209,Z 591.672,A -85,B 0,C 180,E1 11223.156,E2 11223.156} C_VEL
LIN {X 0,Y 246.573,Z 579.842,A -85,B 0,C 180,E1 11218.732,E2 11218.732} C_VEL
LIN {X 0,Y 243.308,Z 570.733,A -85,B 0,C 180,E1 11214.864,E2 11214.864} C_VEL
LIN {X 0,Y 240.456,Z 563.47,A -85,B 0,C 180,E1 11211.411,E2 11211.411} C_VEL
LIN {X 0,Y 238.165,Z 557.559,A -85,B 0,C 180,E1 11208.356,E2 11208.356} C_VEL
LIN {X 0,Y 236.025,Z 553.02,A -85,B 0,C 180,E1 11205.655,E2 11205.655} C_VEL
LIN {X 0,Y 234.734,Z 549.649,A -85,B 0,C 180,E1 11203.446,E2 11203.446} C_VEL
LIN {X 0,Y 234.75,Z 549.543,A -85,B 0,C 180,E1 11198.401,E2 11198.401} C_VEL
LIN {X 0,Y 234.721,Z 549.508,A -85,B 0,C 180,E1 11193.334,E2 11193.334} C_VEL
LIN {X 0,Y 234.752,Z 549.515,A -85,B 0,C 180,E1 11188.16,E2 11188.16} C_VEL
LIN {X 0,Y 234.731,Z 549.538,A -85,B 0,C 180,E1 11183.067,E2 11183.067} C_VEL
LIN {X 0,Y 234.747,Z 549.492,A -85,B 0,C 180,E1 11177.859,E2 11177.859} C_VEL
LIN {X 0,Y 234.737,Z 549.555,A -85,B 0,C 180,E1 11172.738,E2 11172.738} C_VEL
LIN {X 0,Y 234.754,Z 549.496,A -85,B 0,C 180,E1 11167.588,E2 11167.588} C_VEL
LIN {X 0,Y 234.747,Z 549.542,A -85,B 0,C 180,E1 11163.672,E2 11163.672} C_VEL
LIN {X 0,Y 233.918,Z 549.624,A -85,B 0,C 180,E1 11161.924,E2 11161.924} C_VEL
LIN {X 0,Y 230.455,Z 550.075,A -85,B 0,C 180,E1 11159.155,E2 11159.155} C_VEL
LIN {X 0,Y 227.166,Z 550.502,A -85,B 0,C 180,E1 11156.153,E2 11156.153} C_VEL
LIN {X 0,Y 226.82,Z 550.519,A -85,B 0,C 180,E1 11155.02,E2 11155.02} C_VEL
LIN {X 0,Y 226.804,Z 550.519,A -85,B 0,C 180,E1 11149.844,E2 11149.844} C_VEL
LIN {X 0,Y 226.846,Z 550.795,A -85,B 0,C 180,E1 11145.711,E2 11145.711} C_VEL
LIN {X 0,Y 228.651,Z 554.73,A -85,B 0,C 180,E1 11142.964,E2 11142.964} C_VEL
LIN {X 0,Y 231.527,Z 560.935,A -85,B 0,C 180,E1 11139.261,E2 11139.261} C_VEL
LIN {X 0,Y 233.574,Z 565.551,A -85,B 0,C 180,E1 11136.808,E2 11136.808} C_VEL
LIN {X 0,Y 236.356,Z 571.494,A -85,B 0,C 180,E1 11133.9,E2 11133.9} C_VEL
LIN {X 0,Y 240.54,Z 581.95,A -85,B 0,C 180,E1 11129.528,E2 11129.528} C_VEL
LIN {X 0,Y 244.763,Z 593.431,A -85,B 0,C 180,E1 11125.402,E2 11125.402} C_VEL
LIN {X 0,Y 249.37,Z 607.597,A -85,B 0,C 180,E1 11120.987,E2 11120.987} C_VEL
LIN {X 0,Y 253.183,Z 620.447,A -85,B 0,C 180,E1 11117.522,E2 11117.522} C_VEL
LIN {X 0,Y 257.966,Z 630.596,A -85,B 0,C 180,E1 11116.387,E2 11116.387} C_VEL
LIN {X 0,Y 259.728,Z 660.675,A -85,B 0,C 180,E1 11115.103,E2 11115.103} C_VEL
LIN {X 0,Y 253.27,Z 801.678,A -85,B 0,C 180,E1 11111.41,E2 11111.41} C_VEL
LIN {X 0,Y 251.493,Z 819.934,A -85,B 0,C 180,E1 11110.558,E2 11110.558} C_VEL
LIN {X 0,Y 248.81,Z 837.73,A -85,B 0,C 180,E1 11109.34,E2 11109.34} C_VEL
LIN {X 0,Y 245.641,Z 854.579,A -85,B 0,C 180,E1 11107.749,E2 11107.749} C_VEL
LIN {X 0,Y 242.123,Z 870.608,A -85,B 0,C 180,E1 11105.756,E2 11105.756} C_VEL
LIN {X 0,Y 238.433,Z 885.806,A -85,B 0,C 180,E1 11103.322,E2 11103.322} C_VEL
LIN {X 0,Y 234.734,Z 900.011,A -85,B 0,C 180,E1 11100.457,E2 11100.457} C_VEL
LIN {X 0,Y 231.491,Z 912.722,A -85,B 0,C 180,E1 11097.248,E2 11097.248} C_VEL
LIN {X 0,Y 228.777,Z 924.001,A -85,B 0,C 180,E1 11093.71,E2 11093.71} C_VEL
LIN {X 0,Y 226.77,Z 933.86,A -85,B 0,C 180,E1 11089.848,E2 11089.848} C_VEL
LIN {X 0,Y 225.631,Z 942.204,A -85,B 0,C 180,E1 11085.685,E2 11085.685} C_VEL
LIN {X 0,Y 225.395,Z 948.977,A -85,B 0,C 180,E1 11081.258,E2 11081.258} C_VEL
LIN {X 0,Y 225.924,Z 953.804,A -85,B 0,C 180,E1 11076.865,E2 11076.865} C_VEL
LIN {X 0,Y 226.622,Z 956.505,A -85,B 0,C 180,E1 11073.038,E2 11073.038} C_VEL
LIN {X 0,Y 226.84,Z 957.634,A -85,B 0,C 180,E1 11069.751,E2 11069.751} C_VEL
LIN {X 0,Y 226.3,Z 957.55,A -85,B 0,C 180,E1 11066.203,E2 11066.203} C_VEL
LIN {X 0,Y 225.391,Z 955.861,A -85,B 0,C 180,E1 11061.843,E2 11061.843} C_VEL
LIN {X 0,Y 225.026,Z 952.279,A -85,B 0,C 180,E1 11057.168,E2 11057.168} C_VEL
LIN {X 0,Y 225.772,Z 946.864,A -85,B 0,C 180,E1 11052.478,E2 11052.478} C_VEL
LIN {X 0,Y 227.83,Z 939.493,A -85,B 0,C 180,E1 11047.831,E2 11047.831} C_VEL
LIN {X 0,Y 231.106,Z 930.472,A -85,B 0,C 180,E1 11043.543,E2 11043.543} C_VEL
LIN {X 0,Y 235.357,Z 919.914,A -85,B 0,C 180,E1 11039.639,E2 11039.639} C_VEL
LIN {X 0,Y 240.363,Z 907.819,A -85,B 0,C 180,E1 11036.13,E2 11036.13} C_VEL
LIN {X 0,Y 245.753,Z 894.666,A -85,B 0,C 180,E1 11033.129,E2 11033.129} C_VEL
LIN {X 0,Y 251.22,Z 880.193,A -85,B 0,C 180,E1 11030.544,E2 11030.544} C_VEL
LIN {X 0,Y 256.327,Z 865.252,A -85,B 0,C 180,E1 11028.47,E2 11028.47} C_VEL
LIN {X 0,Y 261.152,Z 849.085,A -85,B 0,C 180,E1 11026.747,E2 11026.747} C_VEL
LIN {X 0,Y 265.4,Z 831.949,A -85,B 0,C 180,E1 11025.387,E2 11025.387} C_VEL
LIN {X 0,Y 268.762,Z 814.133,A -85,B 0,C 180,E1 11024.375,E2 11024.375} C_VEL
LIN {X 0,Y 270.901,Z 795.931,A -85,B 0,C 180,E1 11023.687,E2 11023.687} C_VEL
LIN {X 0,Y 279.104,Z 661.033,A -85,B 0,C 180,E1 11020.287,E2 11020.287} C_VEL
LIN {X 0,Y 278.416,Z 649.053,A -85,B 0,C 180,E1 11019.601,E2 11019.601} C_VEL
LIN {X 0,Y 271.819,Z 637.429,A -85,B 0,C 180,E1 11017.235,E2 11017.235} C_VEL
LIN {X 0,Y 265.318,Z 627.172,A -85,B 0,C 180,E1 11014.684,E2 11014.684} C_VEL
LIN {X 0,Y 261.683,Z 621.476,A -85,B 0,C 180,E1 11012.988,E2 11012.988} C_VEL
LIN {X 0,Y 258.825,Z 613.697,A -85,B 0,C 180,E1 11008.874,E2 11008.874} C_VEL
LIN {X 0,Y 256.441,Z 607.717,A -85,B 0,C 180,E1 11004.903,E2 11004.903} C_VEL
LIN {X 0,Y 255.053,Z 604.279,A -85,B 0,C 180,E1 11002.107,E2 11002.107} C_VEL
LIN {X 0,Y 253.533,Z 600.648,A -85,B 0,C 180,E1 10998.39,E2 10998.39} C_VEL
LIN {X 0,Y 251.908,Z 596.821,A -85,B 0,C 180,E1 10992.143,E2 10992.143} C_VEL
LIN {X 0,Y 251.164,Z 596.009,A -85,B 0,C 180,E1 10986.859,E2 10986.859} C_VEL
LIN {X 0,Y 251.417,Z 596.587,A -85,B 0,C 180,E1 10982.051,E2 10982.051} C_VEL
LIN {X 0,Y 252.471,Z 600.228,A -85,B 0,C 180,E1 10975.457,E2 10975.457} C_VEL
LIN {X 0,Y 253.607,Z 603.965,A -85,B 0,C 180,E1 10971.383,E2 10971.383} C_VEL
LIN {X 0,Y 254.825,Z 607.955,A -85,B 0,C 180,E1 10967.997,E2 10967.997} C_VEL
LIN {X 0,Y 256.384,Z 613.102,A -85,B 0,C 180,E1 10964.389,E2 10964.389} C_VEL
LIN {X 0,Y 258.295,Z 620.152,A -85,B 0,C 180,E1 10960.319,E2 10960.319} C_VEL
LIN {X 0,Y 259.764,Z 626.265,A -85,B 0,C 180,E1 10957.361,E2 10957.361} C_VEL
LIN {X 0,Y 265.117,Z 635.99,A -85,B 0,C 180,E1 10954.805,E2 10954.805} C_VEL
LIN {X 0,Y 270.086,Z 645.264,A -85,B 0,C 180,E1 10952.778,E2 10952.778} C_VEL
LIN {X 0,Y 274.036,Z 673.452,A -85,B 0,C 180,E1 10950.37,E2 10950.37} C_VEL
LIN {X 0,Y 275.441,Z 687.035,A -85,B 0,C 180,E1 10949.398,E2 10949.398} C_VEL
LIN {X 0,Y 269.87,Z 769.012,A -85,B 0,C 180,E1 10947.163,E2 10947.163} C_VEL
LIN {X 0,Y 268.063,Z 785.292,A -85,B 0,C 180,E1 10946.366,E2 10946.366} C_VEL
LIN {X 0,Y 265.355,Z 801.252,A -85,B 0,C 180,E1 10945.216,E2 10945.216} C_VEL
LIN {X 0,Y 262.025,Z 815.656,A -85,B 0,C 180,E1 10943.798,E2 10943.798} C_VEL
LIN {X 0,Y 257.823,Z 830.135,A -85,B 0,C 180,E1 10941.919,E2 10941.919} C_VEL
LIN {X 0,Y 253.382,Z 842.805,A -85,B 0,C 180,E1 10939.779,E2 10939.779} C_VEL
LIN {X 0,Y 248.539,Z 854.714,A -85,B 0,C 180,E1 10937.165,E2 10937.165} C_VEL
LIN {X 0,Y 244.136,Z 864.32,A -85,B 0,C 180,E1 10934.445,E2 10934.445} C_VEL
LIN {X 0,Y 239.672,Z 872.972,A -85,B 0,C 180,E1 10931.226,E2 10931.226} C_VEL
LIN {X 0,Y 235.637,Z 880.111,A -85,B 0,C 180,E1 10927.656,E2 10927.656} C_VEL
LIN {X 0,Y 232.277,Z 885.418,A -85,B 0,C 180,E1 10923.819,E2 10923.819} C_VEL
LIN {X 0,Y 229.73,Z 888.991,A -85,B 0,C 180,E1 10919.74,E2 10919.74} C_VEL
LIN {X 0,Y 228.096,Z 890.608,A -85,B 0,C 180,E1 10915.714,E2 10915.714} C_VEL
LIN {X 0,Y 227.203,Z 890.515,A -85,B 0,C 180,E1 10911.418,E2 10911.418} C_VEL
LIN {X 0,Y 227.049,Z 888.703,A -85,B 0,C 180,E1 10907.42,E2 10907.42} C_VEL
LIN {X 0,Y 227.59,Z 884.951,A -85,B 0,C 180,E1 10903.201,E2 10903.201} C_VEL
LIN {X 0,Y 228.775,Z 879.587,A -85,B 0,C 180,E1 10899.302,E2 10899.302} C_VEL
LIN {X 0,Y 230.669,Z 872.259,A -85,B 0,C 180,E1 10895.469,E2 10895.469} C_VEL
LIN {X 0,Y 232.926,Z 864.009,A -85,B 0,C 180,E1 10892.211,E2 10892.211} C_VEL
LIN {X 0,Y 235.736,Z 853.627,A -85,B 0,C 180,E1 10889.025,E2 10889.025} C_VEL
LIN {X 0,Y 238.673,Z 842.174,A -85,B 0,C 180,E1 10886.274,E2 10886.274} C_VEL
LIN {X 0,Y 241.844,Z 828.442,A -85,B 0,C 180,E1 10883.708,E2 10883.708} C_VEL
LIN {X 0,Y 244.546,Z 815.018,A -85,B 0,C 180,E1 10881.77,E2 10881.77} C_VEL
LIN {X 0,Y 247.04,Z 799.859,A -85,B 0,C 180,E1 10880.095,E2 10880.095} C_VEL
LIN {X 0,Y 248.995,Z 784.134,A -85,B 0,C 180,E1 10878.826,E2 10878.826} C_VEL
LIN {X 0,Y 250.398,Z 766.79,A -85,B 0,C 180,E1 10877.89,E2 10877.89} C_VEL
LIN {X 0,Y 254.512,Z 678.214,A -85,B 0,C 180,E1 10875.32,E2 10875.32} C_VEL
LIN {X 0,Y 247.866,Z 627.105,A -85,B 0,C 180,E1 10872.388,E2 10872.388} C_VEL
LIN {X 0,Y 249.294,Z 620.921,A -85,B 0,C 180,E1 10871.041,E2 10871.041} C_VEL
LIN {X 0,Y 246.427,Z 607.356,A -85,B 0,C 180,E1 10866.822,E2 10866.822} C_VEL
LIN {X 0,Y 243.182,Z 594.723,A -85,B 0,C 180,E1 10862.461,E2 10862.461} C_VEL
LIN {X 0,Y 239.88,Z 583.839,A -85,B 0,C 180,E1 10858.246,E2 10858.246} C_VEL
LIN {X 0,Y 236.77,Z 574.974,A -85,B 0,C 180,E1 10854.355,E2 10854.355} C_VEL
LIN {X 0,Y 233.643,Z 566.461,A -85,B 0,C 180,E1 10850.19,E2 10850.19} C_VEL
LIN {X 0,Y 230.27,Z 558.598,A -85,B 0,C 180,E1 10845.647,E2 10845.647} C_VEL
LIN {X 0,Y 228.266,Z 554.245,A -85,B 0,C 180,E1 10842.762,E2 10842.762} C_VEL
LIN {X 0,Y 226.814,Z 550.65,A -85,B 0,C 180,E1 10840.062,E2 10840.062} C_VEL
LIN {X 0,Y 226.791,Z 550.495,A -85,B 0,C 180,E1 10834.662,E2 10834.662} C_VEL
LIN {X 0,Y 226.799,Z 550.539,A -85,B 0,C 180,E1 10829.589,E2 10829.589} C_VEL
LIN {X 0,Y 226.807,Z 550.5,A -85,B 0,C 180,E1 10824.145,E2 10824.145} C_VEL
LIN {X 0,Y 226.8,Z 550.494,A -85,B 0,C 180,E1 10819.308,E2 10819.308} C_VEL
LIN {X 0,Y 226.82,Z 550.538,A -85,B 0,C 180,E1 10813.772,E2 10813.772} C_VEL
LIN {X 0,Y 226.794,Z 550.48,A -85,B 0,C 180,E1 10808.621,E2 10808.621} C_VEL
LIN {X 0,Y 226.811,Z 550.524,A -85,B 0,C 180,E1 10803.539,E2 10803.539} C_VEL
LIN {X 0,Y 226.802,Z 550.498,A -85,B 0,C 180,E1 10798.485,E2 10798.485} C_VEL
LIN {X 0,Y 226.82,Z 550.519,A -85,B 0,C 180,E1 10795.02,E2 10795.02} C_VEL
LIN {X 0,Y 226.018,Z 550.609,A -85,B 0,C 180,E1 10793.893,E2 10793.893} C_VEL
LIN {X 0,Y 221.959,Z 551.095,A -85,B 0,C 180,E1 10791.775,E2 10791.775} C_VEL
LIN {X 0,Y 219.385,Z 551.722,A -85,B 0,C 180,E1 10790.141,E2 10790.141} C_VEL
LIN {X 0,Y 219.093,Z 552.618,A -85,B 0,C 180,E1 10789.203,E2 10789.203} C_VEL
LIN {X 0,Y 221.357,Z 556.96,A -85,B 0,C 180,E1 10785.616,E2 10785.616} C_VEL
LIN {X 0,Y 223.489,Z 561.383,A -85,B 0,C 180,E1 10782.558,E2 10782.558} C_VEL
LIN {X 0,Y 225.777,Z 566.418,A -85,B 0,C 180,E1 10779.522,E2 10779.522} C_VEL
LIN {X 0,Y 228.788,Z 572.96,A -85,B 0,C 180,E1 10775.973,E2 10775.973} C_VEL
LIN {X 0,Y 233.012,Z 583.327,A -85,B 0,C 180,E1 10771.276,E2 10771.276} C_VEL
LIN {X 0,Y 237.296,Z 594.98,A -85,B 0,C 180,E1 10766.787,E2 10766.787} C_VEL
LIN {X 0,Y 241.527,Z 607.87,A -85,B 0,C 180,E1 10762.516,E2 10762.516} C_VEL
LIN {X 0,Y 245.304,Z 620.59,A -85,B 0,C 180,E1 10758.871,E2 10758.871} C_VEL
LIN {X 0,Y 251.562,Z 633.58,A -85,B 0,C 180,E1 10757.322,E2 10757.322} C_VEL
LIN {X 0,Y 253.099,Z 661.527,A -85,B 0,C 180,E1 10756.097,E2 10756.097} C_VEL
LIN {X 0,Y 246.413,Z 801.195,A -85,B 0,C 180,E1 10752.36,E2 10752.36} C_VEL
LIN {X 0,Y 244.566,Z 819.461,A -85,B 0,C 180,E1 10751.486,E2 10751.486} C_VEL
LIN {X 0,Y 241.806,Z 837.145,A -85,B 0,C 180,E1 10750.247,E2 10750.247} C_VEL
LIN {X 0,Y 238.57,Z 853.743,A -85,B 0,C 180,E1 10748.643,E2 10748.643} C_VEL
LIN {X 0,Y 234.881,Z 869.916,A -85,B 0,C 180,E1 10746.581,E2 10746.581} C_VEL
LIN {X 0,Y 231.047,Z 885.074,A -85,B 0,C 180,E1 10744.085,E2 10744.085} C_VEL
LIN {X 0,Y 227.201,Z 899.241,A -85,B 0,C 180,E1 10741.138,E2 10741.138} C_VEL
LIN {X 0,Y 223.7,Z 912.36,A -85,B 0,C 180,E1 10737.701,E2 10737.701} C_VEL
LIN {X 0,Y 220.893,Z 923.524,A -85,B 0,C 180,E1 10734.042,E2 10734.042} C_VEL
LIN {X 0,Y 218.825,Z 933.25,A -85,B 0,C 180,E1 10730.043,E2 10730.043} C_VEL
LIN {X 0,Y 217.663,Z 941.489,A -85,B 0,C 180,E1 10725.727,E2 10725.727} C_VEL
LIN {X 0,Y 217.45,Z 948.165,A -85,B 0,C 180,E1 10721.137,E2 10721.137} C_VEL
LIN {X 0,Y 217.987,Z 952.658,A -85,B 0,C 180,E1 10716.852,E2 10716.852} C_VEL
LIN {X 0,Y 218.728,Z 955.344,A -85,B 0,C 180,E1 10712.885,E2 10712.885} C_VEL
LIN {X 0,Y 218.915,Z 956.449,A -85,B 0,C 180,E1 10709.48,E2 10709.48} C_VEL
LIN {X 0,Y 218.275,Z 956.311,A -85,B 0,C 180,E1 10705.801,E2 10705.801} C_VEL
LIN {X 0,Y 217.348,Z 954.575,A -85,B 0,C 180,E1 10701.272,E2 10701.272} C_VEL
LIN {X 0,Y 217.09,Z 950.904,A -85,B 0,C 180,E1 10696.361,E2 10696.361} C_VEL
LIN {X 0,Y 218.041,Z 945.497,A -85,B 0,C 180,E1 10691.559,E2 10691.559} C_VEL
LIN {X 0,Y 220.401,Z 938.066,A -85,B 0,C 180,E1 10686.76,E2 10686.76} C_VEL
LIN {X 0,Y 224.022,Z 928.983,A -85,B 0,C 180,E1 10682.349,E2 10682.349} C_VEL
LIN {X 0,Y 228.629,Z 918.383,A -85,B 0,C 180,E1 10678.352,E2 10678.352} C_VEL
LIN {X 0,Y 234.018,Z 906.253,A -85,B 0,C 180,E1 10674.782,E2 10674.782} C_VEL
LIN {X 0,Y 239.648,Z 893.203,A -85,B 0,C 180,E1 10671.782,E2 10671.782} C_VEL
LIN {X 0,Y 245.414,Z 878.606,A -85,B 0,C 180,E1 10669.171,E2 10669.171} C_VEL
LIN {X 0,Y 250.882,Z 863.212,A -85,B 0,C 180,E1 10667.048,E2 10667.048} C_VEL
LIN {X 0,Y 255.96,Z 846.662,A -85,B 0,C 180,E1 10665.312,E2 10665.312} C_VEL
LIN {X 0,Y 260.085,Z 830.401,A -85,B 0,C 180,E1 10664.046,E2 10664.046} C_VEL
LIN {X 0,Y 263.487,Z 812.668,A -85,B 0,C 180,E1 10663.054,E2 10663.054} C_VEL
LIN {X 0,Y 265.641,Z 794.504,A -85,B 0,C 180,E1 10662.377,E2 10662.377} C_VEL
LIN {X 0,Y 274.116,Z 662.127,A -85,B 0,C 180,E1 10659.005,E2 10659.005} C_VEL
LIN {X 0,Y 273.629,Z 653.217,A -85,B 0,C 180,E1 10658.476,E2 10658.476} C_VEL
LIN {X 0,Y 267.699,Z 642.634,A -85,B 0,C 180,E1 10656.226,E2 10656.226} C_VEL
LIN {X 0,Y 261.34,Z 632.463,A -85,B 0,C 180,E1 10653.562,E2 10653.562} C_VEL
LIN {X 0,Y 257.217,Z 626.416,A -85,B 0,C 180,E1 10651.653,E2 10651.653} C_VEL
LIN {X 0,Y 254.214,Z 621.741,A -85,B 0,C 180,E1 10649.967,E2 10649.967} C_VEL
LIN {X 0,Y 251.999,Z 615.934,A -85,B 0,C 180,E1 10646.383,E2 10646.383} C_VEL
LIN {X 0,Y 250.008,Z 610.607,A -85,B 0,C 180,E1 10642.329,E2 10642.329} C_VEL
LIN {X 0,Y 248.351,Z 606.731,A -85,B 0,C 180,E1 10638.302,E2 10638.302} C_VEL
LIN {X 0,Y 246.744,Z 602.915,A -85,B 0,C 180,E1 10631.926,E2 10631.926} C_VEL
LIN {X 0,Y 246.024,Z 602.15,A -85,B 0,C 180,E1 10626.534,E2 10626.534} C_VEL
LIN {X 0,Y 246.237,Z 602.703,A -85,B 0,C 180,E1 10622.094,E2 10622.094} C_VEL
LIN {X 0,Y 247.142,Z 606.186,A -85,B 0,C 180,E1 10615.591,E2 10615.591} C_VEL
LIN {X 0,Y 248.203,Z 609.94,A -85,B 0,C 180,E1 10611.428,E2 10611.428} C_VEL
LIN {X 0,Y 249.368,Z 613.943,A -85,B 0,C 180,E1 10607.965,E2 10607.965} C_VEL
LIN {X 0,Y 251.062,Z 619.865,A -85,B 0,C 180,E1 10603.812,E2 10603.812} C_VEL
LIN {X 0,Y 252.589,Z 626.024,A -85,B 0,C 180,E1 10600.338,E2 10600.338} C_VEL
LIN {X 0,Y 257.514,Z 634.537,A -85,B 0,C 180,E1 10597.634,E2 10597.634} C_VEL
LIN {X 0,Y 263.49,Z 645.228,A -85,B 0,C 180,E1 10594.879,E2 10594.879} C_VEL
LIN {X 0,Y 265.902,Z 650.47,A -85,B 0,C 180,E1 10593.824,E2 10593.824} C_VEL
LIN {X 0,Y 269.476,Z 678.324,A -85,B 0,C 180,E1 10591.418,E2 10591.418} C_VEL
LIN {X 0,Y 270.402,Z 688.593,A -85,B 0,C 180,E1 10590.684,E2 10590.684} C_VEL
LIN {X 0,Y 264.658,Z 769.775,A -85,B 0,C 180,E1 10588.454,E2 10588.454} C_VEL
LIN {X 0,Y 262.737,Z 786.164,A -85,B 0,C 180,E1 10587.641,E2 10587.641} C_VEL
LIN {X 0,Y 259.904,Z 802.059,A -85,B 0,C 180,E1 10586.483,E2 10586.483} C_VEL
LIN {X 0,Y 256.29,Z 816.908,A -85,B 0,C 180,E1 10585,E2 10585} C_VEL
LIN {X 0,Y 251.898,Z 831.286,A -85,B 0,C 180,E1 10583.101,E2 10583.101} C_VEL
LIN {X 0,Y 247.234,Z 843.926,A -85,B 0,C 180,E1 10580.929,E2 10580.929} C_VEL
LIN {X 0,Y 242.029,Z 856.085,A -85,B 0,C 180,E1 10578.207,E2 10578.207} C_VEL
LIN {X 0,Y 237.329,Z 865.756,A -85,B 0,C 180,E1 10575.388,E2 10575.388} C_VEL
LIN {X 0,Y 232.632,Z 874.341,A -85,B 0,C 180,E1 10572.096,E2 10572.096} C_VEL
LIN {X 0,Y 228.367,Z 881.421,A -85,B 0,C 180,E1 10568.434,E2 10568.434} C_VEL
LIN {X 0,Y 224.725,Z 886.781,A -85,B 0,C 180,E1 10564.399,E2 10564.399} C_VEL
LIN {X 0,Y 222.063,Z 890.227,A -85,B 0,C 180,E1 10560.278,E2 10560.278} C_VEL
LIN {X 0,Y 220.207,Z 891.864,A -85,B 0,C 180,E1 10555.836,E2 10555.836} C_VEL
LIN {X 0,Y 219.279,Z 891.648,A -85,B 0,C 180,E1 10551.389,E2 10551.389} C_VEL
LIN {X 0,Y 219.146,Z 889.522,A -85,B 0,C 180,E1 10546.973,E2 10546.973} C_VEL
LIN {X 0,Y 219.725,Z 885.867,A -85,B 0,C 180,E1 10542.879,E2 10542.879} C_VEL
LIN {X 0,Y 220.996,Z 880.375,A -85,B 0,C 180,E1 10538.845,E2 10538.845} C_VEL
LIN {X 0,Y 223.017,Z 872.955,A -85,B 0,C 180,E1 10534.883,E2 10534.883} C_VEL
LIN {X 0,Y 225.613,Z 863.842,A -85,B 0,C 180,E1 10531.266,E2 10531.266} C_VEL
LIN {X 0,Y 228.629,Z 853.194,A -85,B 0,C 180,E1 10527.992,E2 10527.992} C_VEL
LIN {X 0,Y 231.895,Z 840.77,A -85,B 0,C 180,E1 10525.05,E2 10525.05} C_VEL
LIN {X 0,Y 234.957,Z 827.889,A -85,B 0,C 180,E1 10522.663,E2 10522.663} C_VEL
LIN {X 0,Y 237.967,Z 813.149,A -85,B 0,C 180,E1 10520.567,E2 10520.567} C_VEL
LIN {X 0,Y 240.417,Z 798.364,A -85,B 0,C 180,E1 10518.969,E2 10518.969} C_VEL
LIN {X 0,Y 242.489,Z 781.283,A -85,B 0,C 180,E1 10517.647,E2 10517.647} C_VEL
LIN {X 0,Y 243.732,Z 764.815,A -85,B 0,C 180,E1 10516.823,E2 10516.823} C_VEL
LIN {X 0,Y 247.884,Z 679.385,A -85,B 0,C 180,E1 10514.319,E2 10514.319} C_VEL
LIN {X 0,Y 241.26,Z 626.919,A -85,B 0,C 180,E1 10511.201,E2 10511.201} C_VEL
LIN {X 0,Y 242.014,Z 623.3,A -85,B 0,C 180,E1 10510.385,E2 10510.385} C_VEL
LIN {X 0,Y 239.331,Z 610.292,A -85,B 0,C 180,E1 10506.196,E2 10506.196} C_VEL
LIN {X 0,Y 236.38,Z 598.494,A -85,B 0,C 180,E1 10501.996,E2 10501.996} C_VEL
LIN {X 0,Y 232.906,Z 586.796,A -85,B 0,C 180,E1 10497.292,E2 10497.292} C_VEL
LIN {X 0,Y 229.738,Z 577.657,A -85,B 0,C 180,E1 10493.087,E2 10493.087} C_VEL
LIN {X 0,Y 226.92,Z 570.416,A -85,B 0,C 180,E1 10489.278,E2 10489.278} C_VEL
LIN {X 0,Y 224.375,Z 563.968,A -85,B 0,C 180,E1 10485.48,E2 10485.48} C_VEL
LIN {X 0,Y 222.323,Z 559.496,A -85,B 0,C 180,E1 10482.424,E2 10482.424} C_VEL
LIN {X 0,Y 220.533,Z 555.528,A -85,B 0,C 180,E1 10479.401,E2 10479.401} C_VEL
LIN {X 0,Y 218.868,Z 551.614,A -85,B 0,C 180,E1 10475.786,E2 10475.786} C_VEL
LIN {X 0,Y 218.873,Z 551.534,A -85,B 0,C 180,E1 10470.303,E2 10470.303} C_VEL
LIN {X 0,Y 218.849,Z 551.478,A -85,B 0,C 180,E1 10465.144,E2 10465.144} C_VEL
LIN {X 0,Y 218.866,Z 551.493,A -85,B 0,C 180,E1 10460.038,E2 10460.038} C_VEL
LIN {X 0,Y 218.852,Z 551.5,A -85,B 0,C 180,E1 10454.824,E2 10454.824} C_VEL
LIN {X 0,Y 218.87,Z 551.467,A -85,B 0,C 180,E1 10449.466,E2 10449.466} C_VEL
LIN {X 0,Y 218.861,Z 551.53,A -85,B 0,C 180,E1 10444.192,E2 10444.192} C_VEL
LIN {X 0,Y 218.88,Z 551.476,A -85,B 0,C 180,E1 10438.954,E2 10438.954} C_VEL
LIN {X 0,Y 218.863,Z 551.487,A -85,B 0,C 180,E1 10433.706,E2 10433.706} C_VEL
LIN {X 0,Y 218.902,Z 551.767,A -85,B 0,C 180,E1 10429.872,E2 10429.872} C_VEL
LIN {X 0,Y 219.093,Z 552.618,A -85,B 0,C 180,E1 10429.203,E2 10429.203} C_VEL
LIN {X 0,Y 219.319,Z 555.805,A -85,B 0,C 180,E1 10427.346,E2 10427.346} C_VEL
LIN {X 0,Y 218.338,Z 567.536,A -85,B 0,C 180,E1 10422.337,E2 10422.337} C_VEL
LIN {X 0,Y 219.117,Z 569.812,A -85,B 0,C 180,E1 10421.019,E2 10421.019} C_VEL
LIN {X 0,Y 221.806,Z 576.06,A -85,B 0,C 180,E1 10417.471,E2 10417.471} C_VEL
LIN {X 0,Y 224.694,Z 582.963,A -85,B 0,C 180,E1 10414.007,E2 10414.007} C_VEL
LIN {X 0,Y 228.246,Z 592.075,A -85,B 0,C 180,E1 10410.041,E2 10410.041} C_VEL
LIN {X 0,Y 232.158,Z 603.416,A -85,B 0,C 180,E1 10405.78,E2 10405.78} C_VEL
LIN {X 0,Y 236.198,Z 616.483,A -85,B 0,C 180,E1 10401.518,E2 10401.518} C_VEL
LIN {X 0,Y 237.527,Z 620.852,A -85,B 0,C 180,E1 10400.299,E2 10400.299} C_VEL
LIN {X 0,Y 245.184,Z 636.47,A -85,B 0,C 180,E1 10398.296,E2 10398.296} C_VEL
LIN {X 0,Y 246.512,Z 662.337,A -85,B 0,C 180,E1 10397.132,E2 10397.132} C_VEL
LIN {X 0,Y 239.625,Z 800.564,A -85,B 0,C 180,E1 10393.365,E2 10393.365} C_VEL
LIN {X 0,Y 237.729,Z 818.765,A -85,B 0,C 180,E1 10392.477,E2 10392.477} C_VEL
LIN {X 0,Y 234.867,Z 836.54,A -85,B 0,C 180,E1 10391.207,E2 10391.207} C_VEL
LIN {X 0,Y 231.517,Z 853.111,A -85,B 0,C 180,E1 10389.569,E2 10389.569} C_VEL
LIN {X 0,Y 227.69,Z 869.224,A -85,B 0,C 180,E1 10387.459,E2 10387.459} C_VEL
LIN {X 0,Y 223.706,Z 884.341,A -85,B 0,C 180,E1 10384.897,E2 10384.897} C_VEL
LIN {X 0,Y 219.55,Z 899.004,A -85,B 0,C 180,E1 10381.736,E2 10381.736} C_VEL
LIN {X 0,Y 215.923,Z 911.997,A -85,B 0,C 180,E1 10378.186,E2 10378.186} C_VEL
LIN {X 0,Y 213.019,Z 923.025,A -85,B 0,C 180,E1 10374.398,E2 10374.398} C_VEL
LIN {X 0,Y 210.832,Z 932.887,A -85,B 0,C 180,E1 10370.116,E2 10370.116} C_VEL
LIN {X 0,Y 209.658,Z 941.196,A -85,B 0,C 180,E1 10365.492,E2 10365.492} C_VEL
LIN {X 0,Y 209.526,Z 947.663,A -85,B 0,C 180,E1 10360.728,E2 10360.728} C_VEL
LIN {X 0,Y 210.151,Z 951.948,A -85,B 0,C 180,E1 10356.285,E2 10356.285} C_VEL
LIN {X 0,Y 210.912,Z 954.411,A -85,B 0,C 180,E1 10352.177,E2 10352.177} C_VEL
LIN {X 0,Y 210.944,Z 955.301,A -85,B 0,C 180,E1 10348.917,E2 10348.917} C_VEL
LIN {X 0,Y 210.166,Z 955.016,A -85,B 0,C 180,E1 10345.091,E2 10345.091} C_VEL
LIN {X 0,Y 209.267,Z 953.137,A -85,B 0,C 180,E1 10340.378,E2 10340.378} C_VEL
LIN {X 0,Y 209.201,Z 949.382,A -85,B 0,C 180,E1 10335.331,E2 10335.331} C_VEL
LIN {X 0,Y 210.474,Z 943.784,A -85,B 0,C 180,E1 10330.294,E2 10330.294} C_VEL
LIN {X 0,Y 213.254,Z 936.148,A -85,B 0,C 180,E1 10325.343,E2 10325.343} C_VEL
LIN {X 0,Y 217.322,Z 926.932,A -85,B 0,C 180,E1 10320.818,E2 10320.818} C_VEL
LIN {X 0,Y 222.383,Z 916.159,A -85,B 0,C 180,E1 10316.741,E2 10316.741} C_VEL
LIN {X 0,Y 227.814,Z 904.688,A -85,B 0,C 180,E1 10313.36,E2 10313.36} C_VEL
LIN {X 0,Y 233.678,Z 891.747,A -85,B 0,C 180,E1 10310.37,E2 10310.37} C_VEL
LIN {X 0,Y 239.603,Z 877.433,A -85,B 0,C 180,E1 10307.799,E2 10307.799} C_VEL
LIN {X 0,Y 245.32,Z 861.992,A -85,B 0,C 180,E1 10305.663,E2 10305.663} C_VEL
LIN {X 0,Y 250.575,Z 845.536,A -85,B 0,C 180,E1 10303.935,E2 10303.935} C_VEL
LIN {X 0,Y 255.055,Z 828.456,A -85,B 0,C 180,E1 10302.617,E2 10302.617} C_VEL
LIN {X 0,Y 258.47,Z 810.708,A -85,B 0,C 180,E1 10301.651,E2 10301.651} C_VEL
LIN {X 0,Y 260.632,Z 792.521,A -85,B 0,C 180,E1 10300.988,E2 10300.988} C_VEL
LIN {X 0,Y 269.269,Z 663.227,A -85,B 0,C 180,E1 10297.676,E2 10297.676} C_VEL
LIN {X 0,Y 268.929,Z 657.328,A -85,B 0,C 180,E1 10297.302,E2 10297.302} C_VEL
LIN {X 0,Y 262.912,Z 646.34,A -85,B 0,C 180,E1 10294.848,E2 10294.848} C_VEL
LIN {X 0,Y 255.669,Z 634.797,A -85,B 0,C 180,E1 10291.524,E2 10291.524} C_VEL
LIN {X 0,Y 249.824,Z 626.666,A -85,B 0,C 180,E1 10288.442,E2 10288.442} C_VEL
LIN {X 0,Y 246.818,Z 622.247,A -85,B 0,C 180,E1 10286.462,E2 10286.462} C_VEL
LIN {X 0,Y 244.833,Z 616.728,A -85,B 0,C 180,E1 10282.321,E2 10282.321} C_VEL
LIN {X 0,Y 243.173,Z 612.817,A -85,B 0,C 180,E1 10278.209,E2 10278.209} C_VEL
LIN {X 0,Y 241.636,Z 609.075,A -85,B 0,C 180,E1 10271.94,E2 10271.94} C_VEL
LIN {X 0,Y 240.897,Z 608.293,A -85,B 0,C 180,E1 10266.434,E2 10266.434} C_VEL
LIN {X 0,Y 241.061,Z 608.824,A -85,B 0,C 180,E1 10262.139,E2 10262.139} C_VEL
LIN {X 0,Y 241.829,Z 612.156,A -85,B 0,C 180,E1 10255.731,E2 10255.731} C_VEL
LIN {X 0,Y 242.746,Z 615.663,A -85,B 0,C 180,E1 10251.711,E2 10251.711} C_VEL
LIN {X 0,Y 243.83,Z 619.654,A -85,B 0,C 180,E1 10248.168,E2 10248.168} C_VEL
LIN {X 0,Y 245.427,Z 625.552,A -85,B 0,C 180,E1 10243.977,E2 10243.977} C_VEL
LIN {X 0,Y 250.08,Z 633.362,A -85,B 0,C 180,E1 10240.861,E2 10240.861} C_VEL
LIN {X 0,Y 255.114,Z 642.143,A -85,B 0,C 180,E1 10238.14,E2 10238.14} C_VEL
LIN {X 0,Y 260.146,Z 651.452,A -85,B 0,C 180,E1 10235.716,E2 10235.716} C_VEL
LIN {X 0,Y 261.748,Z 655.237,A -85,B 0,C 180,E1 10234.957,E2 10234.957} C_VEL
LIN {X 0,Y 264.902,Z 682.242,A -85,B 0,C 180,E1 10232.581,E2 10232.581} C_VEL
LIN {X 0,Y 265.515,Z 690.029,A -85,B 0,C 180,E1 10232.021,E2 10232.021} C_VEL
LIN {X 0,Y 259.601,Z 770.325,A -85,B 0,C 180,E1 10229.803,E2 10229.803} C_VEL
LIN {X 0,Y 257.626,Z 786.595,A -85,B 0,C 180,E1 10228.997,E2 10228.997} C_VEL
LIN {X 0,Y 254.592,Z 802.936,A -85,B 0,C 180,E1 10227.802,E2 10227.802} C_VEL
LIN {X 0,Y 250.958,Z 817.305,A -85,B 0,C 180,E1 10226.364,E2 10226.364} C_VEL
LIN {X 0,Y 246.358,Z 831.773,A -85,B 0,C 180,E1 10224.451,E2 10224.451} C_VEL
LIN {X 0,Y 241.467,Z 844.519,A -85,B 0,C 180,E1 10222.257,E2 10222.257} C_VEL
LIN {X 0,Y 236.202,Z 856.239,A -85,B 0,C 180,E1 10219.626,E2 10219.626} C_VEL
LIN {X 0,Y 231.003,Z 866.473,A -85,B 0,C 180,E1 10216.639,E2 10216.639} C_VEL
LIN {X 0,Y 226.004,Z 875.125,A -85,B 0,C 180,E1 10213.284,E2 10213.284} C_VEL
LIN {X 0,Y 221.435,Z 882.294,A -85,B 0,C 180,E1 10209.535,E2 10209.535} C_VEL
LIN {X 0,Y 217.674,Z 887.526,A -85,B 0,C 180,E1 10205.606,E2 10205.606} C_VEL
LIN {X 0,Y 214.575,Z 891.28,A -85,B 0,C 180,E1 10201.14,E2 10201.14} C_VEL
LIN {X 0,Y 212.606,Z 892.985,A -85,B 0,C 180,E1 10196.832,E2 10196.832} C_VEL
LIN {X 0,Y 211.442,Z 892.927,A -85,B 0,C 180,E1 10192.051,E2 10192.051} C_VEL
LIN {X 0,Y 211.191,Z 891.081,A -85,B 0,C 180,E1 10187.633,E2 10187.633} C_VEL
LIN {X 0,Y 211.734,Z 887.332,A -85,B 0,C 180,E1 10183.096,E2 10183.096} C_VEL
LIN {X 0,Y 213,Z 882.001,A -85,B 0,C 180,E1 10178.907,E2 10178.907} C_VEL
LIN {X 0,Y 215.044,Z 874.711,A -85,B 0,C 180,E1 10174.797,E2 10174.797} C_VEL
LIN {X 0,Y 217.488,Z 866.557,A -85,B 0,C 180,E1 10171.314,E2 10171.314} C_VEL
LIN {X 0,Y 220.528,Z 856.264,A -85,B 0,C 180,E1 10167.918,E2 10167.918} C_VEL
LIN {X 0,Y 223.713,Z 844.997,A -85,B 0,C 180,E1 10164.997,E2 10164.997} C_VEL
LIN {X 0,Y 226.971,Z 832.144,A -85,B 0,C 180,E1 10162.403,E2 10162.403} C_VEL
LIN {X 0,Y 230.059,Z 818.417,A -85,B 0,C 180,E1 10160.239,E2 10160.239} C_VEL
LIN {X 0,Y 232.759,Z 803.726,A -85,B 0,C 180,E1 10158.476,E2 10158.476} C_VEL
LIN {X 0,Y 235.073,Z 787.461,A -85,B 0,C 180,E1 10157.033,E2 10157.033} C_VEL
LIN {X 0,Y 236.645,Z 770.592,A -85,B 0,C 180,E1 10156.031,E2 10156.031} C_VEL
LIN {X 0,Y 238.143,Z 741.939,A -85,B 0,C 180,E1 10155.065,E2 10155.065} C_VEL
LIN {X 0,Y 241.284,Z 680.421,A -85,B 0,C 180,E1 10153.269,E2 10153.269} C_VEL
LIN {X 0,Y 234.712,Z 627.155,A -85,B 0,C 180,E1 10150.008,E2 10150.008} C_VEL
LIN {X 0,Y 234.701,Z 625.256,A -85,B 0,C 180,E1 10149.552,E2 10149.552} C_VEL
LIN {X 0,Y 232.096,Z 612.572,A -85,B 0,C 180,E1 10145.299,E2 10145.299} C_VEL
LIN {X 0,Y 229.281,Z 601.105,A -85,B 0,C 180,E1 10141.049,E2 10141.049} C_VEL
LIN {X 0,Y 226.076,Z 590.142,A -85,B 0,C 180,E1 10136.438,E2 10136.438} C_VEL
LIN {X 0,Y 222.949,Z 581.162,A -85,B 0,C 180,E1 10132.091,E2 10132.091} C_VEL
LIN {X 0,Y 220.004,Z 573.055,A -85,B 0,C 180,E1 10127.626,E2 10127.626} C_VEL
LIN {X 0,Y 217.916,Z 568.367,A -85,B 0,C 180,E1 10124.589,E2 10124.589} C_VEL
LIN {X 0,Y 216.302,Z 564.582,A -85,B 0,C 180,E1 10121.908,E2 10121.908} C_VEL
LIN {X 0,Y 214.874,Z 561.159,A -85,B 0,C 180,E1 10119.261,E2 10119.261} C_VEL
LIN {X 0,Y 212.72,Z 556.66,A -85,B 0,C 180,E1 10115.13,E2 10115.13} C_VEL
LIN {X 0,Y 210.942,Z 552.613,A -85,B 0,C 180,E1 10110.384,E2 10110.384} C_VEL
LIN {X 0,Y 210.909,Z 552.467,A -85,B 0,C 180,E1 10104.957,E2 10104.957} C_VEL
LIN {X 0,Y 210.93,Z 552.472,A -85,B 0,C 180,E1 10099.668,E2 10099.668} C_VEL
LIN {X 0,Y 210.932,Z 552.505,A -85,B 0,C 180,E1 10093.99,E2 10093.99} C_VEL
LIN {X 0,Y 210.917,Z 552.454,A -85,B 0,C 180,E1 10088.726,E2 10088.726} C_VEL
LIN {X 0,Y 210.933,Z 552.49,A -85,B 0,C 180,E1 10083.261,E2 10083.261} C_VEL
LIN {X 0,Y 210.923,Z 552.484,A -85,B 0,C 180,E1 10077.827,E2 10077.827} C_VEL
LIN {X 0,Y 210.985,Z 552.813,A -85,B 0,C 180,E1 10075.243,E2 10075.243} C_VEL
LIN {X 0,Y 213.508,Z 558.01,A -85,B 0,C 180,E1 10069.75,E2 10069.75} C_VEL
LIN {X 0,Y 215.853,Z 562.793,A -85,B 0,C 180,E1 10065.789,E2 10065.789} C_VEL
LIN {X 0,Y 217.924,Z 567.344,A -85,B 0,C 180,E1 10062.611,E2 10062.611} C_VEL
LIN {X 0,Y 219.117,Z 569.812,A -85,B 0,C 180,E1 10061.019,E2 10061.019} C_VEL
LIN {X 0,Y 219.945,Z 572.745,A -85,B 0,C 180,E1 10059.486,E2 10059.486} C_VEL
LIN {X 0,Y 219.698,Z 577.931,A -85,B 0,C 180,E1 10057.595,E2 10057.595} C_VEL
LIN {X 0,Y 219.01,Z 587.734,A -85,B 0,C 180,E1 10054.338,E2 10054.338} C_VEL
LIN {X 0,Y 219.53,Z 590.132,A -85,B 0,C 180,E1 10053.346,E2 10053.346} C_VEL
LIN {X 0,Y 223.221,Z 600.369,A -85,B 0,C 180,E1 10048.996,E2 10048.996} C_VEL
LIN {X 0,Y 226.961,Z 611.878,A -85,B 0,C 180,E1 10044.753,E2 10044.753} C_VEL
LIN {X 0,Y 229.71,Z 620.977,A -85,B 0,C 180,E1 10041.864,E2 10041.864} C_VEL
LIN {X 0,Y 238.864,Z 639.174,A -85,B 0,C 180,E1 10039.331,E2 10039.331} C_VEL
LIN {X 0,Y 240.001,Z 663.159,A -85,B 0,C 180,E1 10038.22,E2 10038.22} C_VEL
LIN {X 0,Y 232.878,Z 799.991,A -85,B 0,C 180,E1 10034.413,E2 10034.413} C_VEL
LIN {X 0,Y 230.904,Z 818.273,A -85,B 0,C 180,E1 10033.5,E2 10033.5} C_VEL
LIN {X 0,Y 227.997,Z 835.731,A -85,B 0,C 180,E1 10032.226,E2 10032.226} C_VEL
LIN {X 0,Y 224.527,Z 852.314,A -85,B 0,C 180,E1 10030.554,E2 10030.554} C_VEL
LIN {X 0,Y 220.559,Z 868.439,A -85,B 0,C 180,E1 10028.394,E2 10028.394} C_VEL
LIN {X 0,Y 216.412,Z 883.557,A -85,B 0,C 180,E1 10025.765,E2 10025.765} C_VEL
LIN {X 0,Y 212.083,Z 898.216,A -85,B 0,C 180,E1 10022.511,E2 10022.511} C_VEL
LIN {X 0,Y 208.414,Z 910.736,A -85,B 0,C 180,E1 10018.984,E2 10018.984} C_VEL
LIN {X 0,Y 205.339,Z 921.81,A -85,B 0,C 180,E1 10015.065,E2 10015.065} C_VEL
LIN {X 0,Y 203.012,Z 931.654,A -85,B 0,C 180,E1 10010.648,E2 10010.648} C_VEL
LIN {X 0,Y 201.732,Z 940.019,A -85,B 0,C 180,E1 10005.821,E2 10005.821} C_VEL
LIN {X 0,Y 201.569,Z 946.525,A -85,B 0,C 180,E1 10000.842,E2 10000.842} C_VEL
LIN {X 0,Y 202.22,Z 950.783,A -85,B 0,C 180,E1 9996.248,E2 9996.248} C_VEL
LIN {X 0,Y 202.988,Z 953.123,A -85,B 0,C 180,E1 9992.262,E2 9992.262} C_VEL
LIN {X 0,Y 203.069,Z 954.008,A -85,B 0,C 180,E1 9989.157,E2 9989.157} C_VEL
LIN {X 0,Y 202.249,Z 953.883,A -85,B 0,C 180,E1 9985.183,E2 9985.183} C_VEL
LIN {X 0,Y 201.299,Z 952.154,A -85,B 0,C 180,E1 9980.282,E2 9980.282} C_VEL
LIN {X 0,Y 201.256,Z 948.547,A -85,B 0,C 180,E1 9975.033,E2 9975.033} C_VEL
LIN {X 0,Y 202.63,Z 943.118,A -85,B 0,C 180,E1 9969.799,E2 9969.799} C_VEL
LIN {X 0,Y 205.592,Z 935.743,A -85,B 0,C 180,E1 9964.667,E2 9964.667} C_VEL
LIN {X 0,Y 209.888,Z 926.708,A -85,B 0,C 180,E1 9959.994,E2 9959.994} C_VEL
LIN {X 0,Y 215.234,Z 916.067,A -85,B 0,C 180,E1 9955.78,E2 9955.78} C_VEL
LIN {X 0,Y 221.317,Z 903.995,A -85,B 0,C 180,E1 9952.098,E2 9952.098} C_VEL
LIN {X 0,Y 227.674,Z 890.723,A -85,B 0,C 180,E1 9948.971,E2 9948.971} C_VEL
LIN {X 0,Y 233.974,Z 876.258,A -85,B 0,C 180,E1 9946.349,E2 9946.349} C_VEL
LIN {X 0,Y 239.915,Z 860.91,A -85,B 0,C 180,E1 9944.217,E2 9944.217} C_VEL
LIN {X 0,Y 245.386,Z 844.41,A -85,B 0,C 180,E1 9942.49,E2 9942.49} C_VEL
LIN {X 0,Y 250.032,Z 827.225,A -85,B 0,C 180,E1 9941.177,E2 9941.177} C_VEL
LIN {X 0,Y 253.535,Z 809.369,A -85,B 0,C 180,E1 9940.217,E2 9940.217} C_VEL
LIN {X 0,Y 255.756,Z 790.883,A -85,B 0,C 180,E1 9939.554,E2 9939.554} C_VEL
LIN {X 0,Y 264.572,Z 664.261,A -85,B 0,C 180,E1 9936.295,E2 9936.295} C_VEL
LIN {X 0,Y 264.366,Z 661.427,A -85,B 0,C 180,E1 9936.09,E2 9936.09} C_VEL
LIN {X 0,Y 258.379,Z 650.594,A -85,B 0,C 180,E1 9933.465,E2 9933.465} C_VEL
LIN {X 0,Y 252.392,Z 640.904,A -85,B 0,C 180,E1 9930.535,E2 9930.535} C_VEL
LIN {X 0,Y 247.531,Z 633.826,A -85,B 0,C 180,E1 9927.812,E2 9927.812} C_VEL
LIN {X 0,Y 243.232,Z 627.926,A -85,B 0,C 180,E1 9925.049,E2 9925.049} C_VEL
LIN {X 0,Y 239.572,Z 622.68,A -85,B 0,C 180,E1 9922.062,E2 9922.062} C_VEL
LIN {X 0,Y 237.881,Z 618.75,A -85,B 0,C 180,E1 9917.868,E2 9917.868} C_VEL
LIN {X 0,Y 236.477,Z 615.169,A -85,B 0,C 180,E1 9911.709,E2 9911.709} C_VEL
LIN {X 0,Y 235.76,Z 614.427,A -85,B 0,C 180,E1 9906.086,E2 9906.086} C_VEL
LIN {X 0,Y 235.88,Z 614.941,A -85,B 0,C 180,E1 9902.186,E2 9902.186} C_VEL
LIN {X 0,Y 236.529,Z 618.137,A -85,B 0,C 180,E1 9895.879,E2 9895.879} C_VEL
LIN {X 0,Y 237.354,Z 621.644,A -85,B 0,C 180,E1 9891.765,E2 9891.765} C_VEL
LIN {X 0,Y 238.397,Z 625.457,A -85,B 0,C 180,E1 9888.386,E2 9888.386} C_VEL
LIN {X 0,Y 243.758,Z 634.086,A -85,B 0,C 180,E1 9884.048,E2 9884.048} C_VEL
LIN {X 0,Y 248.39,Z 641.832,A -85,B 0,C 180,E1 9881.092,E2 9881.092} C_VEL
LIN {X 0,Y 252.344,Z 648.982,A -85,B 0,C 180,E1 9878.864,E2 9878.864} C_VEL
LIN {X 0,Y 256.911,Z 657.788,A -85,B 0,C 180,E1 9876.55,E2 9876.55} C_VEL
LIN {X 0,Y 257.761,Z 660.255,A -85,B 0,C 180,E1 9876.101,E2 9876.101} C_VEL
LIN {X 0,Y 260.549,Z 687.149,A -85,B 0,C 180,E1 9873.704,E2 9873.704} C_VEL
LIN {X 0,Y 260.763,Z 691.656,A -85,B 0,C 180,E1 9873.403,E2 9873.403} C_VEL
LIN {X 0,Y 254.685,Z 770.982,A -85,B 0,C 180,E1 9871.202,E2 9871.202} C_VEL
LIN {X 0,Y 252.624,Z 787.276,A -85,B 0,C 180,E1 9870.391,E2 9870.391} C_VEL
LIN {X 0,Y 249.565,Z 803.145,A -85,B 0,C 180,E1 9869.233,E2 9869.233} C_VEL
LIN {X 0,Y 245.775,Z 817.702,A -85,B 0,C 180,E1 9867.785,E2 9867.785} C_VEL
LIN {X 0,Y 240.99,Z 832.182,A -85,B 0,C 180,E1 9865.874,E2 9865.874} C_VEL
LIN {X 0,Y 235.839,Z 845.12,A -85,B 0,C 180,E1 9863.649,E2 9863.649} C_VEL
LIN {X 0,Y 230.275,Z 856.951,A -85,B 0,C 180,E1 9860.979,E2 9860.979} C_VEL
LIN {X 0,Y 224.801,Z 867.219,A -85,B 0,C 180,E1 9857.958,E2 9857.958} C_VEL
LIN {X 0,Y 219.487,Z 875.951,A -85,B 0,C 180,E1 9854.541,E2 9854.541} C_VEL
LIN {X 0,Y 214.593,Z 883.171,A -85,B 0,C 180,E1 9850.707,E2 9850.707} C_VEL
LIN {X 0,Y 210.465,Z 888.577,A -85,B 0,C 180,E1 9846.594,E2 9846.594} C_VEL
LIN {X 0,Y 207.138,Z 892.329,A -85,B 0,C 180,E1 9842.064,E2 9842.064} C_VEL
LIN {X 0,Y 204.95,Z 894.152,A -85,B 0,C 180,E1 9837.604,E2 9837.604} C_VEL
LIN {X 0,Y 203.634,Z 894.201,A -85,B 0,C 180,E1 9832.818,E2 9832.818} C_VEL
LIN {X 0,Y 203.258,Z 892.598,A -85,B 0,C 180,E1 9828.302,E2 9828.302} C_VEL
LIN {X 0,Y 203.69,Z 889.079,A -85,B 0,C 180,E1 9823.623,E2 9823.623} C_VEL
LIN {X 0,Y 204.894,Z 884.015,A -85,B 0,C 180,E1 9819.263,E2 9819.263} C_VEL
LIN {X 0,Y 206.81,Z 877.328,A -85,B 0,C 180,E1 9815.155,E2 9815.155} C_VEL
LIN {X 0,Y 209.566,Z 868.478,A -85,B 0,C 180,E1 9811.09,E2 9811.09} C_VEL
LIN {X 0,Y 212.691,Z 858.421,A -85,B 0,C 180,E1 9807.572,E2 9807.572} C_VEL
LIN {X 0,Y 216.271,Z 846.339,A -85,B 0,C 180,E1 9804.293,E2 9804.293} C_VEL
LIN {X 0,Y 219.663,Z 833.599,A -85,B 0,C 180,E1 9801.622,E2 9801.622} C_VEL
LIN {X 0,Y 223.06,Z 819.16,A -85,B 0,C 180,E1 9799.277,E2 9799.277} C_VEL
LIN {X 0,Y 225.878,Z 804.445,A -85,B 0,C 180,E1 9797.471,E2 9797.471} C_VEL
LIN {X 0,Y 228.293,Z 788.168,A -85,B 0,C 180,E1 9795.995,E2 9795.995} C_VEL
LIN {X 0,Y 229.938,Z 771.32,A -85,B 0,C 180,E1 9794.971,E2 9794.971} C_VEL
LIN {X 0,Y 231.475,Z 743.194,A -85,B 0,C 180,E1 9793.998,E2 9793.998} C_VEL
LIN {X 0,Y 234.758,Z 681.398,A -85,B 0,C 180,E1 9792.157,E2 9792.157} C_VEL
LIN {X 0,Y 228.484,Z 629.473,A -85,B 0,C 180,E1 9788.869,E2 9788.869} C_VEL
LIN {X 0,Y 227.356,Z 626.764,A -85,B 0,C 180,E1 9788.455,E2 9788.455} C_VEL
LIN {X 0,Y 224.713,Z 613.912,A -85,B 0,C 180,E1 9784.002,E2 9784.002} C_VEL
LIN {X 0,Y 221.968,Z 602.966,A -85,B 0,C 180,E1 9779.701,E2 9779.701} C_VEL
LIN {X 0,Y 219.066,Z 592.878,A -85,B 0,C 180,E1 9775.242,E2 9775.242} C_VEL
LIN {X 0,Y 215.874,Z 583.61,A -85,B 0,C 180,E1 9770.46,E2 9770.46} C_VEL
LIN {X 0,Y 213.291,Z 576.858,A -85,B 0,C 180,E1 9766.441,E2 9766.441} C_VEL
LIN {X 0,Y 211.064,Z 570.948,A -85,B 0,C 180,E1 9762.459,E2 9762.459} C_VEL
LIN {X 0,Y 208.96,Z 566.42,A -85,B 0,C 180,E1 9758.745,E2 9758.745} C_VEL
LIN {X 0,Y 207.088,Z 562.283,A -85,B 0,C 180,E1 9754.837,E2 9754.837} C_VEL
LIN {X 0,Y 205.102,Z 558.034,A -85,B 0,C 180,E1 9749.805,E2 9749.805} C_VEL
LIN {X 0,Y 203.026,Z 553.683,A -85,B 0,C 180,E1 9741.677,E2 9741.677} C_VEL
LIN {X 0,Y 202.985,Z 553.452,A -85,B 0,C 180,E1 9736.013,E2 9736.013} C_VEL
LIN {X 0,Y 202.978,Z 553.457,A -85,B 0,C 180,E1 9730.789,E2 9730.789} C_VEL
LIN {X 0,Y 203.007,Z 553.555,A -85,B 0,C 180,E1 9725.37,E2 9725.37} C_VEL
LIN {X 0,Y 203.281,Z 554.846,A -85,B 0,C 180,E1 9721.974,E2 9721.974} C_VEL
LIN {X 0,Y 205.664,Z 558.915,A -85,B 0,C 180,E1 9715.26,E2 9715.26} C_VEL
LIN {X 0,Y 208.056,Z 563.78,A -85,B 0,C 180,E1 9710.038,E2 9710.038} C_VEL
LIN {X 0,Y 210.336,Z 568.609,A -85,B 0,C 180,E1 9705.97,E2 9705.97} C_VEL
LIN {X 0,Y 212.339,Z 573.149,A -85,B 0,C 180,E1 9702.744,E2 9702.744} C_VEL
LIN {X 0,Y 214.244,Z 577.329,A -85,B 0,C 180,E1 9700.082,E2 9700.082} C_VEL
LIN {X 0,Y 217.261,Z 584.504,A -85,B 0,C 180,E1 9696.11,E2 9696.11} C_VEL
LIN {X 0,Y 219.53,Z 590.132,A -85,B 0,C 180,E1 9693.346,E2 9693.346} C_VEL
LIN {X 0,Y 220.152,Z 593.882,A -85,B 0,C 180,E1 9691.921,E2 9691.921} C_VEL
LIN {X 0,Y 219.531,Z 601.369,A -85,B 0,C 180,E1 9689.756,E2 9689.756} C_VEL
LIN {X 0,Y 218.907,Z 609.835,A -85,B 0,C 180,E1 9687.382,E2 9687.382} C_VEL
LIN {X 0,Y 219.517,Z 613.23,A -85,B 0,C 180,E1 9686.23,E2 9686.23} C_VEL
LIN {X 0,Y 221.945,Z 621.158,A -85,B 0,C 180,E1 9683.552,E2 9683.552} C_VEL
LIN {X 0,Y 231.213,Z 639.182,A -85,B 0,C 180,E1 9680.81,E2 9680.81} C_VEL
LIN {X 0,Y 232.677,Z 642.711,A -85,B 0,C 180,E1 9680.378,E2 9680.378} C_VEL
LIN {X 0,Y 233.586,Z 663.905,A -85,B 0,C 180,E1 9679.371,E2 9679.371} C_VEL
LIN {X 0,Y 226.229,Z 799.246,A -85,B 0,C 180,E1 9675.531,E2 9675.531} C_VEL
LIN {X 0,Y 224.204,Z 817.436,A -85,B 0,C 180,E1 9674.607,E2 9674.607} C_VEL
LIN {X 0,Y 221.19,Z 835.003,A -85,B 0,C 180,E1 9673.3,E2 9673.3} C_VEL
LIN {X 0,Y 217.608,Z 851.504,A -85,B 0,C 180,E1 9671.601,E2 9671.601} C_VEL
LIN {X 0,Y 213.517,Z 867.518,A -85,B 0,C 180,E1 9669.407,E2 9669.407} C_VEL
LIN {X 0,Y 209.171,Z 882.718,A -85,B 0,C 180,E1 9666.692,E2 9666.692} C_VEL
LIN {X 0,Y 204.659,Z 897.357,A -85,B 0,C 180,E1 9663.341,E2 9663.341} C_VEL
LIN {X 0,Y 200.683,Z 910.309,A -85,B 0,C 180,E1 9659.555,E2 9659.555} C_VEL
LIN {X 0,Y 197.493,Z 921.257,A -85,B 0,C 180,E1 9655.49,E2 9655.49} C_VEL
LIN {X 0,Y 195.128,Z 930.783,A -85,B 0,C 180,E1 9651.022,E2 9651.022} C_VEL
LIN {X 0,Y 193.81,Z 938.841,A -85,B 0,C 180,E1 9646.178,E2 9646.178} C_VEL
LIN {X 0,Y 193.607,Z 945.327,A -85,B 0,C 180,E1 9641.019,E2 9641.019} C_VEL
LIN {X 0,Y 194.289,Z 949.618,A -85,B 0,C 180,E1 9636.207,E2 9636.207} C_VEL
LIN {X 0,Y 195.1,Z 951.95,A -85,B 0,C 180,E1 9632.059,E2 9632.059} C_VEL
LIN {X 0,Y 195.119,Z 952.809,A -85,B 0,C 180,E1 9628.829,E2 9628.829} C_VEL
LIN {X 0,Y 194.187,Z 952.634,A -85,B 0,C 180,E1 9624.686,E2 9624.686} C_VEL
LIN {X 0,Y 193.249,Z 950.793,A -85,B 0,C 180,E1 9619.434,E2 9619.434} C_VEL
LIN {X 0,Y 193.453,Z 946.986,A -85,B 0,C 180,E1 9613.799,E2 9613.799} C_VEL
LIN {X 0,Y 195.208,Z 941.432,A -85,B 0,C 180,E1 9608.365,E2 9608.365} C_VEL
LIN {X 0,Y 198.417,Z 934.354,A -85,B 0,C 180,E1 9603.36,E2 9603.36} C_VEL
LIN {X 0,Y 203.13,Z 925.271,A -85,B 0,C 180,E1 9598.557,E2 9598.557} C_VEL
LIN {X 0,Y 208.874,Z 914.641,A -85,B 0,C 180,E1 9594.275,E2 9594.275} C_VEL
LIN {X 0,Y 214.937,Z 903.352,A -85,B 0,C 180,E1 9590.762,E2 9590.762} C_VEL
LIN {X 0,Y 221.609,Z 890.211,A -85,B 0,C 180,E1 9587.592,E2 9587.592} C_VEL
LIN {X 0,Y 228.16,Z 875.946,A -85,B 0,C 180,E1 9584.958,E2 9584.958} C_VEL
LIN {X 0,Y 234.368,Z 860.645,A -85,B 0,C 180,E1 9582.805,E2 9582.805} C_VEL
LIN {X 0,Y 240.037,Z 844.293,A -85,B 0,C 180,E1 9581.077,E2 9581.077} C_VEL
LIN {X 0,Y 244.667,Z 827.985,A -85,B 0,C 180,E1 9579.81,E2 9579.81} C_VEL
LIN {X 0,Y 248.417,Z 810.253,A -85,B 0,C 180,E1 9578.823,E2 9578.823} C_VEL
LIN {X 0,Y 250.791,Z 792.199,A -85,B 0,C 180,E1 9578.151,E2 9578.151} C_VEL
LIN {X 0,Y 260.058,Z 665.944,A -85,B 0,C 180,E1 9574.883,E2 9574.883} C_VEL
LIN {X 0,Y 254.738,Z 656.101,A -85,B 0,C 180,E1 9572.396,E2 9572.396} C_VEL
LIN {X 0,Y 249.394,Z 647.238,A -85,B 0,C 180,E1 9569.612,E2 9569.612} C_VEL
LIN {X 0,Y 245.086,Z 640.74,A -85,B 0,C 180,E1 9567.057,E2 9567.057} C_VEL
LIN {X 0,Y 241.182,Z 635.196,A -85,B 0,C 180,E1 9564.426,E2 9564.426} C_VEL
LIN {X 0,Y 237.127,Z 629.69,A -85,B 0,C 180,E1 9561.131,E2 9561.131} C_VEL
LIN {X 0,Y 233.374,Z 625.199,A -85,B 0,C 180,E1 9557.323,E2 9557.323} C_VEL
LIN {X 0,Y 231.693,Z 622.669,A -85,B 0,C 180,E1 9554.239,E2 9554.239} C_VEL
LIN {X 0,Y 231.241,Z 621.159,A -85,B 0,C 180,E1 9551.073,E2 9551.073} C_VEL
LIN {X 0,Y 230.635,Z 620.574,A -85,B 0,C 180,E1 9545.223,E2 9545.223} C_VEL
LIN {X 0,Y 230.697,Z 621.182,A -85,B 0,C 180,E1 9541.987,E2 9541.987} C_VEL
LIN {X 0,Y 231.238,Z 624.122,A -85,B 0,C 180,E1 9536.032,E2 9536.032} C_VEL
LIN {X 0,Y 232.729,Z 627.227,A -85,B 0,C 180,E1 9532.966,E2 9532.966} C_VEL
LIN {X 0,Y 237.253,Z 634.177,A -85,B 0,C 180,E1 9528.205,E2 9528.205} C_VEL
LIN {X 0,Y 241.608,Z 641.311,A -85,B 0,C 180,E1 9524.703,E2 9524.703} C_VEL
LIN {X 0,Y 245.831,Z 648.638,A -85,B 0,C 180,E1 9521.871,E2 9521.871} C_VEL
LIN {X 0,Y 249.529,Z 655.631,A -85,B 0,C 180,E1 9519.659,E2 9519.659} C_VEL
LIN {X 0,Y 253.754,Z 664.207,A -85,B 0,C 180,E1 9517.392,E2 9517.392} C_VEL
LIN {X 0,Y 256.212,Z 690.641,A -85,B 0,C 180,E1 9514.995,E2 9514.995} C_VEL
LIN {X 0,Y 256.155,Z 694.249,A -85,B 0,C 180,E1 9514.819,E2 9514.819} C_VEL
LIN {X 0,Y 249.957,Z 771.762,A -85,B 0,C 180,E1 9512.657,E2 9512.657} C_VEL
LIN {X 0,Y 247.783,Z 788.101,A -85,B 0,C 180,E1 9511.838,E2 9511.838} C_VEL
LIN {X 0,Y 244.536,Z 804.156,A -85,B 0,C 180,E1 9510.657,E2 9510.657} C_VEL
LIN {X 0,Y 240.448,Z 819.046,A -85,B 0,C 180,E1 9509.156,E2 9509.156} C_VEL
LIN {X 0,Y 235.433,Z 833.512,A -85,B 0,C 180,E1 9507.221,E2 9507.221} C_VEL
LIN {X 0,Y 230.109,Z 846.245,A -85,B 0,C 180,E1 9505,E2 9505} C_VEL
LIN {X 0,Y 224.463,Z 857.705,A -85,B 0,C 180,E1 9502.391,E2 9502.391} C_VEL
LIN {X 0,Y 218.724,Z 867.955,A -85,B 0,C 180,E1 9499.351,E2 9499.351} C_VEL
LIN {X 0,Y 213.087,Z 876.786,A -85,B 0,C 180,E1 9495.873,E2 9495.873} C_VEL
LIN {X 0,Y 207.854,Z 884.069,A -85,B 0,C 180,E1 9491.953,E2 9491.953} C_VEL
LIN {X 0,Y 203.538,Z 889.428,A -85,B 0,C 180,E1 9487.875,E2 9487.875} C_VEL
LIN {X 0,Y 199.961,Z 893.201,A -85,B 0,C 180,E1 9483.361,E2 9483.361} C_VEL
LIN {X 0,Y 197.334,Z 895.307,A -85,B 0,C 180,E1 9478.436,E2 9478.436} C_VEL
LIN {X 0,Y 195.826,Z 895.447,A -85,B 0,C 180,E1 9473.463,E2 9473.463} C_VEL
LIN {X 0,Y 195.333,Z 893.805,A -85,B 0,C 180,E1 9468.498,E2 9468.498} C_VEL
LIN {X 0,Y 195.705,Z 890.544,A -85,B 0,C 180,E1 9463.889,E2 9463.889} C_VEL
LIN {X 0,Y 197.002,Z 885.2,A -85,B 0,C 180,E1 9459.048,E2 9459.048} C_VEL
LIN {X 0,Y 198.932,Z 878.752,A -85,B 0,C 180,E1 9454.898,E2 9454.898} C_VEL
LIN {X 0,Y 201.646,Z 870.372,A -85,B 0,C 180,E1 9450.849,E2 9450.849} C_VEL
LIN {X 0,Y 204.863,Z 860.579,A -85,B 0,C 180,E1 9447.199,E2 9447.199} C_VEL
LIN {X 0,Y 208.535,Z 848.743,A -85,B 0,C 180,E1 9443.809,E2 9443.809} C_VEL
LIN {X 0,Y 212.051,Z 836.412,A -85,B 0,C 180,E1 9441.046,E2 9441.046} C_VEL
LIN {X 0,Y 215.58,Z 822.237,A -85,B 0,C 180,E1 9438.604,E2 9438.604} C_VEL
LIN {X 0,Y 218.678,Z 807.419,A -85,B 0,C 180,E1 9436.648,E2 9436.648} C_VEL
LIN {X 0,Y 221.286,Z 791.076,A -85,B 0,C 180,E1 9435.073,E2 9435.073} C_VEL
LIN {X 0,Y 223.11,Z 774.709,A -85,B 0,C 180,E1 9433.979,E2 9433.979} C_VEL
LIN {X 0,Y 224.398,Z 753.194,A -85,B 0,C 180,E1 9433.142,E2 9433.142} C_VEL
LIN {X 0,Y 228.343,Z 682.494,A -85,B 0,C 180,E1 9430.989,E2 9430.989} C_VEL
LIN {X 0,Y 222.574,Z 632.811,A -85,B 0,C 180,E1 9427.731,E2 9427.731} C_VEL
LIN {X 0,Y 219.76,Z 626.735,A -85,B 0,C 180,E1 9426.79,E2 9426.79} C_VEL
LIN {X 0,Y 217.183,Z 614.469,A -85,B 0,C 180,E1 9422.29,E2 9422.29} C_VEL
LIN {X 0,Y 214.549,Z 604.025,A -85,B 0,C 180,E1 9417.908,E2 9417.908} C_VEL
LIN {X 0,Y 211.803,Z 594.774,A -85,B 0,C 180,E1 9413.501,E2 9413.501} C_VEL
LIN {X 0,Y 208.886,Z 586.131,A -85,B 0,C 180,E1 9408.721,E2 9408.721} C_VEL
LIN {X 0,Y 206.27,Z 579.283,A -85,B 0,C 180,E1 9404.269,E2 9404.269} C_VEL
LIN {X 0,Y 204.581,Z 575.205,A -85,B 0,C 180,E1 9401.18,E2 9401.18} C_VEL
LIN {X 0,Y 203.16,Z 571.812,A -85,B 0,C 180,E1 9398.325,E2 9398.325} C_VEL
LIN {X 0,Y 201.477,Z 567.919,A -85,B 0,C 180,E1 9394.534,E2 9394.534} C_VEL
LIN {X 0,Y 199.719,Z 563.945,A -85,B 0,C 180,E1 9389.712,E2 9389.712} C_VEL
LIN {X 0,Y 197.632,Z 559.553,A -85,B 0,C 180,E1 9381.363,E2 9381.363} C_VEL
LIN {X 0,Y 196.753,Z 558.485,A -85,B 0,C 180,E1 9375.089,E2 9375.089} C_VEL
LIN {X 0,Y 196.97,Z 558.728,A -85,B 0,C 180,E1 9368.76,E2 9368.76} C_VEL
LIN {X 0,Y 197.816,Z 559.917,A -85,B 0,C 180,E1 9364.058,E2 9364.058} C_VEL
LIN {X 0,Y 200.358,Z 564.917,A -85,B 0,C 180,E1 9355.421,E2 9355.421} C_VEL
LIN {X 0,Y 202.588,Z 569.531,A -85,B 0,C 180,E1 9350.34,E2 9350.34} C_VEL
LIN {X 0,Y 204.813,Z 574.414,A -85,B 0,C 180,E1 9346.161,E2 9346.161} C_VEL
LIN {X 0,Y 206.783,Z 579.003,A -85,B 0,C 180,E1 9342.846,E2 9342.846} C_VEL
LIN {X 0,Y 208.647,Z 583.227,A -85,B 0,C 180,E1 9340.109,E2 9340.109} C_VEL
LIN {X 0,Y 212.087,Z 591.535,A -85,B 0,C 180,E1 9335.485,E2 9335.485} C_VEL
LIN {X 0,Y 215.702,Z 601.464,A -85,B 0,C 180,E1 9330.876,E2 9330.876} C_VEL
LIN {X 0,Y 219.269,Z 612.472,A -85,B 0,C 180,E1 9326.513,E2 9326.513} C_VEL
LIN {X 0,Y 219.517,Z 613.23,A -85,B 0,C 180,E1 9326.23,E2 9326.23} C_VEL
LIN {X 0,Y 220.585,Z 617.747,A -85,B 0,C 180,E1 9325.007,E2 9325.007} C_VEL
LIN {X 0,Y 221.656,Z 625.272,A -85,B 0,C 180,E1 9323.807,E2 9323.807} C_VEL
LIN {X 0,Y 224.032,Z 638.732,A -85,B 0,C 180,E1 9322.344,E2 9322.344} C_VEL
LIN {X 0,Y 225.749,Z 643.646,A -85,B 0,C 180,E1 9321.755,E2 9321.755} C_VEL
LIN {X 0,Y 226.554,Z 646.075,A -85,B 0,C 180,E1 9321.487,E2 9321.487} C_VEL
LIN {X 0,Y 227.269,Z 664.649,A -85,B 0,C 180,E1 9320.585,E2 9320.585} C_VEL
LIN {X 0,Y 219.655,Z 798.673,A -85,B 0,C 180,E1 9316.709,E2 9316.709} C_VEL
LIN {X 0,Y 217.561,Z 816.824,A -85,B 0,C 180,E1 9315.766,E2 9315.766} C_VEL
LIN {X 0,Y 214.499,Z 834.111,A -85,B 0,C 180,E1 9314.457,E2 9314.457} C_VEL
LIN {X 0,Y 210.766,Z 850.694,A -85,B 0,C 180,E1 9312.717,E2 9312.717} C_VEL
LIN {X 0,Y 206.489,Z 866.796,A -85,B 0,C 180,E1 9310.455,E2 9310.455} C_VEL
LIN {X 0,Y 201.97,Z 881.943,A -85,B 0,C 180,E1 9307.673,E2 9307.673} C_VEL
LIN {X 0,Y 197.281,Z 896.496,A -85,B 0,C 180,E1 9304.235,E2 9304.235} C_VEL
LIN {X 0,Y 193.248,Z 908.973,A -85,B 0,C 180,E1 9300.469,E2 9300.469} C_VEL
LIN {X 0,Y 189.863,Z 919.988,A -85,B 0,C 180,E1 9296.256,E2 9296.256} C_VEL
LIN {X 0,Y 187.332,Z 929.547,A -85,B 0,C 180,E1 9291.612,E2 9291.612} C_VEL
LIN {X 0,Y 185.898,Z 937.636,A -85,B 0,C 180,E1 9286.565,E2 9286.565} C_VEL
LIN {X 0,Y 185.647,Z 944.146,A -85,B 0,C 180,E1 9281.183,E2 9281.183} C_VEL
LIN {X 0,Y 186.356,Z 948.448,A -85,B 0,C 180,E1 9276.163,E2 9276.163} C_VEL
LIN {X 0,Y 187.215,Z 950.775,A -85,B 0,C 180,E1 9271.84,E2 9271.84} C_VEL
LIN {X 0,Y 187.202,Z 951.56,A -85,B 0,C 180,E1 9268.78,E2 9268.78} C_VEL
LIN {X 0,Y 186.188,Z 951.443,A -85,B 0,C 180,E1 9264.457,E2 9264.457} C_VEL
LIN {X 0,Y 185.263,Z 949.735,A -85,B 0,C 180,E1 9259.117,E2 9259.117} C_VEL
LIN {X 0,Y 185.595,Z 945.921,A -85,B 0,C 180,E1 9253.093,E2 9253.093} C_VEL
LIN {X 0,Y 187.585,Z 940.433,A -85,B 0,C 180,E1 9247.439,E2 9247.439} C_VEL
LIN {X 0,Y 191.261,Z 933.145,A -85,B 0,C 180,E1 9242.065,E2 9242.065} C_VEL
LIN {X 0,Y 196.332,Z 924.178,A -85,B 0,C 180,E1 9237.171,E2 9237.171} C_VEL
LIN {X 0,Y 202.282,Z 913.94,A -85,B 0,C 180,E1 9232.921,E2 9232.921} C_VEL
LIN {X 0,Y 209.18,Z 901.862,A -85,B 0,C 180,E1 9229.101,E2 9229.101} C_VEL
LIN {X 0,Y 216.27,Z 888.536,A -85,B 0,C 180,E1 9225.89,E2 9225.89} C_VEL
LIN {X 0,Y 222.978,Z 874.515,A -85,B 0,C 180,E1 9223.319,E2 9223.319} C_VEL
LIN {X 0,Y 229.285,Z 859.561,A -85,B 0,C 180,E1 9221.226,E2 9221.226} C_VEL
LIN {X 0,Y 235.179,Z 843.166,A -85,B 0,C 180,E1 9219.509,E2 9219.509} C_VEL
LIN {X 0,Y 240.143,Z 826.181,A -85,B 0,C 180,E1 9218.209,E2 9218.209} C_VEL
LIN {X 0,Y 243.9,Z 808.543,A -85,B 0,C 180,E1 9217.256,E2 9217.256} C_VEL
LIN {X 0,Y 246.298,Z 790.459,A -85,B 0,C 180,E1 9216.597,E2 9216.597} C_VEL
LIN {X 0,Y 255.573,Z 669.724,A -85,B 0,C 180,E1 9213.478,E2 9213.478} C_VEL
LIN {X 0,Y 250.094,Z 659.619,A -85,B 0,C 180,E1 9210.712,E2 9210.712} C_VEL
LIN {X 0,Y 245.487,Z 651.897,A -85,B 0,C 180,E1 9208.062,E2 9208.062} C_VEL
LIN {X 0,Y 240.335,Z 644.03,A -85,B 0,C 180,E1 9204.649,E2 9204.649} C_VEL
LIN {X 0,Y 235.475,Z 637.258,A -85,B 0,C 180,E1 9200.636,E2 9200.636} C_VEL
LIN {X 0,Y 231.991,Z 632.916,A -85,B 0,C 180,E1 9196.93,E2 9196.93} C_VEL
LIN {X 0,Y 228.797,Z 628.939,A -85,B 0,C 180,E1 9191.831,E2 9191.831} C_VEL
LIN {X 0,Y 227.218,Z 627.806,A -85,B 0,C 180,E1 9186.062,E2 9186.062} C_VEL
LIN {X 0,Y 227.349,Z 628.248,A -85,B 0,C 180,E1 9182.52,E2 9182.52} C_VEL
LIN {X 0,Y 229.508,Z 631.911,A -85,B 0,C 180,E1 9176.253,E2 9176.253} C_VEL
LIN {X 0,Y 231.842,Z 635.934,A -85,B 0,C 180,E1 9172.69,E2 9172.69} C_VEL
LIN {X 0,Y 235.467,Z 641.617,A -85,B 0,C 180,E1 9168.798,E2 9168.798} C_VEL
LIN {X 0,Y 239.491,Z 648.533,A -85,B 0,C 180,E1 9165.369,E2 9165.369} C_VEL
LIN {X 0,Y 243.318,Z 655.444,A -85,B 0,C 180,E1 9162.667,E2 9162.667} C_VEL
LIN {X 0,Y 247.806,Z 664.202,A -85,B 0,C 180,E1 9159.881,E2 9159.881} C_VEL
LIN {X 0,Y 249.978,Z 669.34,A -85,B 0,C 180,E1 9158.608,E2 9158.608} C_VEL
LIN {X 0,Y 251.962,Z 693.812,A -85,B 0,C 180,E1 9156.366,E2 9156.366} C_VEL
LIN {X 0,Y 245.442,Z 772.328,A -85,B 0,C 180,E1 9154.179,E2 9154.179} C_VEL
LIN {X 0,Y 243.177,Z 788.726,A -85,B 0,C 180,E1 9153.359,E2 9153.359} C_VEL
LIN {X 0,Y 239.71,Z 805.177,A -85,B 0,C 180,E1 9152.147,E2 9152.147} C_VEL
LIN {X 0,Y 235.59,Z 819.596,A -85,B 0,C 180,E1 9150.695,E2 9150.695} C_VEL
LIN {X 0,Y 230.351,Z 834.097,A -85,B 0,C 180,E1 9148.756,E2 9148.756} C_VEL
LIN {X 0,Y 224.769,Z 846.901,A -85,B 0,C 180,E1 9146.522,E2 9146.522} C_VEL
LIN {X 0,Y 218.805,Z 858.457,A -85,B 0,C 180,E1 9143.879,E2 9143.879} C_VEL
LIN {X 0,Y 212.786,Z 868.691,A -85,B 0,C 180,E1 9140.823,E2 9140.823} C_VEL
LIN {X 0,Y 206.812,Z 877.62,A -85,B 0,C 180,E1 9137.285,E2 9137.285} C_VEL
LIN {X 0,Y 201.221,Z 884.966,A -85,B 0,C 180,E1 9133.282,E2 9133.282} C_VEL
LIN {X 0,Y 196.573,Z 890.404,A -85,B 0,C 180,E1 9129.095,E2 9129.095} C_VEL
LIN {X 0,Y 192.634,Z 894.303,A -85,B 0,C 180,E1 9124.381,E2 9124.381} C_VEL
LIN {X 0,Y 189.759,Z 896.445,A -85,B 0,C 180,E1 9119.335,E2 9119.335} C_VEL
LIN {X 0,Y 188.119,Z 896.745,A -85,B 0,C 180,E1 9114.486,E2 9114.486} C_VEL
LIN {X 0,Y 187.419,Z 895.229,A -85,B 0,C 180,E1 9109.215,E2 9109.215} C_VEL
LIN {X 0,Y 187.721,Z 892.001,A -85,B 0,C 180,E1 9104.177,E2 9104.177} C_VEL
LIN {X 0,Y 188.998,Z 886.76,A -85,B 0,C 180,E1 9099.127,E2 9099.127} C_VEL
LIN {X 0,Y 190.957,Z 880.48,A -85,B 0,C 180,E1 9094.802,E2 9094.802} C_VEL
LIN {X 0,Y 193.731,Z 872.26,A -85,B 0,C 180,E1 9090.588,E2 9090.588} C_VEL
LIN {X 0,Y 197.038,Z 862.659,A -85,B 0,C 180,E1 9086.797,E2 9086.797} C_VEL
LIN {X 0,Y 200.669,Z 851.623,A -85,B 0,C 180,E1 9083.417,E2 9083.417} C_VEL
LIN {X 0,Y 204.635,Z 838.455,A -85,B 0,C 180,E1 9080.293,E2 9080.293} C_VEL
LIN {X 0,Y 208.261,Z 824.781,A -85,B 0,C 180,E1 9077.802,E2 9077.802} C_VEL
LIN {X 0,Y 211.725,Z 809.172,A -85,B 0,C 180,E1 9075.643,E2 9075.643} C_VEL
LIN {X 0,Y 214.345,Z 793.953,A -85,B 0,C 180,E1 9074.093,E2 9074.093} C_VEL
LIN {X 0,Y 216.445,Z 776.702,A -85,B 0,C 180,E1 9072.863,E2 9072.863} C_VEL
LIN {X 0,Y 217.67,Z 758.362,A -85,B 0,C 180,E1 9072.082,E2 9072.082} C_VEL
LIN {X 0,Y 221.992,Z 683.443,A -85,B 0,C 180,E1 9069.749,E2 9069.749} C_VEL
LIN {X 0,Y 216.75,Z 636.217,A -85,B 0,C 180,E1 9066.551,E2 9066.551} C_VEL
LIN {X 0,Y 212.051,Z 626.279,A -85,B 0,C 180,E1 9064.868,E2 9064.868} C_VEL
LIN {X 0,Y 209.594,Z 614.65,A -85,B 0,C 180,E1 9060.254,E2 9060.254} C_VEL
LIN {X 0,Y 206.782,Z 603.737,A -85,B 0,C 180,E1 9055.287,E2 9055.287} C_VEL
LIN {X 0,Y 203.922,Z 594.447,A -85,B 0,C 180,E1 9050.336,E2 9050.336} C_VEL
LIN {X 0,Y 201.073,Z 586.518,A -85,B 0,C 180,E1 9045.324,E2 9045.324} C_VEL
LIN {X 0,Y 198.891,Z 580.828,A -85,B 0,C 180,E1 9041.056,E2 9041.056} C_VEL
LIN {X 0,Y 197.519,Z 577.447,A -85,B 0,C 180,E1 9038.14,E2 9038.14} C_VEL
LIN {X 0,Y 195.891,Z 573.579,A -85,B 0,C 180,E1 9034.222,E2 9034.222} C_VEL
LIN {X 0,Y 194.192,Z 569.683,A -85,B 0,C 180,E1 9029.285,E2 9029.285} C_VEL
LIN {X 0,Y 192.343,Z 565.531,A -85,B 0,C 180,E1 9021.02,E2 9021.02} C_VEL
LIN {X 0,Y 191.574,Z 564.591,A -85,B 0,C 180,E1 9014.818,E2 9014.818} C_VEL
LIN {X 0,Y 191.882,Z 564.926,A -85,B 0,C 180,E1 9008.39,E2 9008.39} C_VEL
LIN {X 0,Y 192.674,Z 566.153,A -85,B 0,C 180,E1 9003.869,E2 9003.869} C_VEL
LIN {X 0,Y 195.045,Z 570.909,A -85,B 0,C 180,E1 8995.59,E2 8995.59} C_VEL
LIN {X 0,Y 197.207,Z 575.621,A -85,B 0,C 180,E1 8990.369,E2 8990.369} C_VEL
LIN {X 0,Y 199.155,Z 579.809,A -85,B 0,C 180,E1 8986.648,E2 8986.648} C_VEL
LIN {X 0,Y 201.231,Z 584.831,A -85,B 0,C 180,E1 8982.954,E2 8982.954} C_VEL
LIN {X 0,Y 203.586,Z 590.183,A -85,B 0,C 180,E1 8979.443,E2 8979.443} C_VEL
LIN {X 0,Y 207.24,Z 599.808,A -85,B 0,C 180,E1 8974.265,E2 8974.265} C_VEL
LIN {X 0,Y 210.621,Z 609.79,A -85,B 0,C 180,E1 8969.765,E2 8969.765} C_VEL
LIN {X 0,Y 214.125,Z 621.142,A -85,B 0,C 180,E1 8965.435,E2 8965.435} C_VEL
LIN {X 0,Y 222.901,Z 637.83,A -85,B 0,C 180,E1 8962.61,E2 8962.61} C_VEL
LIN {X 0,Y 225.749,Z 643.646,A -85,B 0,C 180,E1 8961.755,E2 8961.755} C_VEL
LIN {X 0,Y 226.705,Z 647.569,A -85,B 0,C 180,E1 8961.395,E2 8961.395} C_VEL
LIN {X 0,Y 226.565,Z 652.958,A -85,B 0,C 180,E1 8961.203,E2 8961.203} C_VEL
LIN {X 0,Y 224.837,Z 660.601,A -85,B 0,C 180,E1 8961.246,E2 8961.246} C_VEL
LIN {X 0,Y 221.036,Z 673.19,A -85,B 0,C 180,E1 8961.521,E2 8961.521} C_VEL
LIN {X 0,Y 220.16,Z 679.055,A -85,B 0,C 180,E1 8961.462,E2 8961.462} C_VEL
LIN {X 0,Y 213.161,Z 798.027,A -85,B 0,C 180,E1 8957.951,E2 8957.951} C_VEL
LIN {X 0,Y 210.992,Z 816.208,A -85,B 0,C 180,E1 8956.991,E2 8956.991} C_VEL
LIN {X 0,Y 207.745,Z 833.9,A -85,B 0,C 180,E1 8955.62,E2 8955.62} C_VEL
LIN {X 0,Y 203.754,Z 850.883,A -85,B 0,C 180,E1 8953.782,E2 8953.782} C_VEL
LIN {X 0,Y 199.328,Z 866.746,A -85,B 0,C 180,E1 8951.463,E2 8951.463} C_VEL
LIN {X 0,Y 194.664,Z 881.679,A -85,B 0,C 180,E1 8948.614,E2 8948.614} C_VEL
LIN {X 0,Y 189.941,Z 895.677,A -85,B 0,C 180,E1 8945.185,E2 8945.185} C_VEL
LIN {X 0,Y 185.574,Z 908.525,A -85,B 0,C 180,E1 8941.149,E2 8941.149} C_VEL
LIN {X 0,Y 182.051,Z 919.404,A -85,B 0,C 180,E1 8936.769,E2 8936.769} C_VEL
LIN {X 0,Y 179.418,Z 928.868,A -85,B 0,C 180,E1 8931.926,E2 8931.926} C_VEL
LIN {X 0,Y 177.937,Z 936.865,A -85,B 0,C 180,E1 8926.656,E2 8926.656} C_VEL
LIN {X 0,Y 177.687,Z 942.951,A -85,B 0,C 180,E1 8921.362,E2 8921.362} C_VEL
LIN {X 0,Y 178.423,Z 947.265,A -85,B 0,C 180,E1 8916.115,E2 8916.115} C_VEL
LIN {X 0,Y 179.332,Z 949.593,A -85,B 0,C 180,E1 8911.601,E2 8911.601} C_VEL
LIN {X 0,Y 179.285,Z 950.306,A -85,B 0,C 180,E1 8908.726,E2 8908.726} C_VEL
LIN {X 0,Y 178.184,Z 950.251,A -85,B 0,C 180,E1 8904.207,E2 8904.207} C_VEL
LIN {X 0,Y 177.271,Z 948.605,A -85,B 0,C 180,E1 8898.62,E2 8898.62} C_VEL
LIN {X 0,Y 177.691,Z 945.104,A -85,B 0,C 180,E1 8892.654,E2 8892.654} C_VEL
LIN {X 0,Y 180.016,Z 939.438,A -85,B 0,C 180,E1 8886.434,E2 8886.434} C_VEL
LIN {X 0,Y 184.137,Z 932.097,A -85,B 0,C 180,E1 8880.752,E2 8880.752} C_VEL
LIN {X 0,Y 189.678,Z 923.081,A -85,B 0,C 180,E1 8875.673,E2 8875.673} C_VEL
LIN {X 0,Y 196.264,Z 912.51,A -85,B 0,C 180,E1 8871.208,E2 8871.208} C_VEL
LIN {X 0,Y 203.091,Z 901.242,A -85,B 0,C 180,E1 8867.595,E2 8867.595} C_VEL
LIN {X 0,Y 210.471,Z 888.11,A -85,B 0,C 180,E1 8864.37,E2 8864.37} C_VEL
LIN {X 0,Y 217.652,Z 873.858,A -85,B 0,C 180,E1 8861.722,E2 8861.722} C_VEL
LIN {X 0,Y 224.394,Z 858.566,A -85,B 0,C 180,E1 8859.58,E2 8859.58} C_VEL
LIN {X 0,Y 230.513,Z 842.201,A -85,B 0,C 180,E1 8857.879,E2 8857.879} C_VEL
LIN {X 0,Y 235.64,Z 825.184,A -85,B 0,C 180,E1 8856.592,E2 8856.592} C_VEL
LIN {X 0,Y 239.492,Z 807.55,A -85,B 0,C 180,E1 8855.654,E2 8855.654} C_VEL
LIN {X 0,Y 241.965,Z 789.298,A -85,B 0,C 180,E1 8854.999,E2 8854.999} C_VEL
LIN {X 0,Y 251.189,Z 673.677,A -85,B 0,C 180,E1 8852.011,E2 8852.011} C_VEL
LIN {X 0,Y 245.96,Z 663.8,A -85,B 0,C 180,E1 8849.109,E2 8849.109} C_VEL
LIN {X 0,Y 240.829,Z 655.293,A -85,B 0,C 180,E1 8845.844,E2 8845.844} C_VEL
LIN {X 0,Y 237.009,Z 649.416,A -85,B 0,C 180,E1 8842.968,E2 8842.968} C_VEL
LIN {X 0,Y 233.714,Z 644.696,A -85,B 0,C 180,E1 8840.014,E2 8840.014} C_VEL
LIN {X 0,Y 230.501,Z 640.493,A -85,B 0,C 180,E1 8836.376,E2 8836.376} C_VEL
LIN {X 0,Y 227.578,Z 636.738,A -85,B 0,C 180,E1 8831.402,E2 8831.402} C_VEL
LIN {X 0,Y 226.166,Z 635.72,A -85,B 0,C 180,E1 8825.581,E2 8825.581} C_VEL
LIN {X 0,Y 226.321,Z 636.242,A -85,B 0,C 180,E1 8822.532,E2 8822.532} C_VEL
LIN {X 0,Y 228.329,Z 639.801,A -85,B 0,C 180,E1 8816.485,E2 8816.485} C_VEL
LIN {X 0,Y 230.505,Z 643.769,A -85,B 0,C 180,E1 8813.023,E2 8813.023} C_VEL
LIN {X 0,Y 233.649,Z 648.932,A -85,B 0,C 180,E1 8809.458,E2 8809.458} C_VEL
LIN {X 0,Y 237.369,Z 655.616,A -85,B 0,C 180,E1 8806.107,E2 8806.107} C_VEL
LIN {X 0,Y 240.854,Z 662.248,A -85,B 0,C 180,E1 8803.479,E2 8803.479} C_VEL
LIN {X 0,Y 245.028,Z 670.81,A -85,B 0,C 180,E1 8800.73,E2 8800.73} C_VEL
LIN {X 0,Y 246.327,Z 674.21,A -85,B 0,C 180,E1 8799.894,E2 8799.894} C_VEL
LIN {X 0,Y 247.767,Z 695.596,A -85,B 0,C 180,E1 8797.905,E2 8797.905} C_VEL
LIN {X 0,Y 241.101,Z 772.945,A -85,B 0,C 180,E1 8795.756,E2 8795.756} C_VEL
LIN {X 0,Y 238.752,Z 789.336,A -85,B 0,C 180,E1 8794.939,E2 8794.939} C_VEL
LIN {X 0,Y 235.199,Z 805.604,A -85,B 0,C 180,E1 8793.748,E2 8793.748} C_VEL
LIN {X 0,Y 230.912,Z 820.147,A -85,B 0,C 180,E1 8792.296,E2 8792.296} C_VEL
LIN {X 0,Y 225.446,Z 834.709,A -85,B 0,C 180,E1 8790.358,E2 8790.358} C_VEL
LIN {X 0,Y 219.614,Z 847.567,A -85,B 0,C 180,E1 8788.12,E2 8788.12} C_VEL
LIN {X 0,Y 213.33,Z 859.247,A -85,B 0,C 180,E1 8785.45,E2 8785.45} C_VEL
LIN {X 0,Y 207.005,Z 869.48,A -85,B 0,C 180,E1 8782.374,E2 8782.374} C_VEL
LIN {X 0,Y 200.675,Z 878.473,A -85,B 0,C 180,E1 8778.784,E2 8778.784} C_VEL
LIN {X 0,Y 194.708,Z 885.864,A -85,B 0,C 180,E1 8774.7,E2 8774.7} C_VEL
LIN {X 0,Y 189.385,Z 891.71,A -85,B 0,C 180,E1 8770.089,E2 8770.089} C_VEL
LIN {X 0,Y 185.218,Z 895.525,A -85,B 0,C 180,E1 8765.275,E2 8765.275} C_VEL
LIN {X 0,Y 182.078,Z 897.672,A -85,B 0,C 180,E1 8759.974,E2 8759.974} C_VEL
LIN {X 0,Y 180.205,Z 897.891,A -85,B 0,C 180,E1 8754.584,E2 8754.584} C_VEL
LIN {X 0,Y 179.493,Z 896.306,A -85,B 0,C 180,E1 8749.181,E2 8749.181} C_VEL
LIN {X 0,Y 179.784,Z 893.166,A -85,B 0,C 180,E1 8744.159,E2 8744.159} C_VEL
LIN {X 0,Y 181.104,Z 887.92,A -85,B 0,C 180,E1 8738.888,E2 8738.888} C_VEL
LIN {X 0,Y 183.326,Z 881.118,A -85,B 0,C 180,E1 8734.062,E2 8734.062} C_VEL
LIN {X 0,Y 186.289,Z 872.775,A -85,B 0,C 180,E1 8729.689,E2 8729.689} C_VEL
LIN {X 0,Y 189.803,Z 863.057,A -85,B 0,C 180,E1 8725.767,E2 8725.767} C_VEL
LIN {X 0,Y 193.787,Z 851.39,A -85,B 0,C 180,E1 8722.16,E2 8722.16} C_VEL
LIN {X 0,Y 197.825,Z 838.519,A -85,B 0,C 180,E1 8719.072,E2 8719.072} C_VEL
LIN {X 0,Y 201.636,Z 824.583,A -85,B 0,C 180,E1 8716.52,E2 8716.52} C_VEL
LIN {X 0,Y 205.049,Z 809.753,A -85,B 0,C 180,E1 8714.441,E2 8714.441} C_VEL
LIN {X 0,Y 207.786,Z 794.457,A -85,B 0,C 180,E1 8712.857,E2 8712.857} C_VEL
LIN {X 0,Y 209.968,Z 777.254,A -85,B 0,C 180,E1 8711.608,E2 8711.608} C_VEL
LIN {X 0,Y 211.258,Z 758.736,A -85,B 0,C 180,E1 8710.808,E2 8710.808} C_VEL
LIN {X 0,Y 215.738,Z 684.549,A -85,B 0,C 180,E1 8708.459,E2 8708.459} C_VEL
LIN {X 0,Y 211.028,Z 639.843,A -85,B 0,C 180,E1 8705.32,E2 8705.32} C_VEL
LIN {X 0,Y 204.507,Z 626.167,A -85,B 0,C 180,E1 8702.852,E2 8702.852} C_VEL
LIN {X 0,Y 202.295,Z 616.083,A -85,B 0,C 180,E1 8698.57,E2 8698.57} C_VEL
LIN {X 0,Y 199.981,Z 606.818,A -85,B 0,C 180,E1 8694.093,E2 8694.093} C_VEL
LIN {X 0,Y 197.23,Z 597.923,A -85,B 0,C 180,E1 8689.057,E2 8689.057} C_VEL
LIN {X 0,Y 194.742,Z 590.389,A -85,B 0,C 180,E1 8684.045,E2 8684.045} C_VEL
LIN {X 0,Y 192.757,Z 585.446,A -85,B 0,C 180,E1 8680.032,E2 8680.032} C_VEL
LIN {X 0,Y 191.693,Z 582.724,A -85,B 0,C 180,E1 8677.55,E2 8677.55} C_VEL
LIN {X 0,Y 190.308,Z 579.236,A -85,B 0,C 180,E1 8673.89,E2 8673.89} C_VEL
LIN {X 0,Y 188.78,Z 575.548,A -85,B 0,C 180,E1 8669.085,E2 8669.085} C_VEL
LIN {X 0,Y 187.128,Z 571.596,A -85,B 0,C 180,E1 8660.978,E2 8660.978} C_VEL
LIN {X 0,Y 186.419,Z 570.706,A -85,B 0,C 180,E1 8654.919,E2 8654.919} C_VEL
LIN {X 0,Y 186.755,Z 571.072,A -85,B 0,C 180,E1 8648.312,E2 8648.312} C_VEL
LIN {X 0,Y 187.496,Z 572.252,A -85,B 0,C 180,E1 8643.976,E2 8643.976} C_VEL
LIN {X 0,Y 189.664,Z 576.615,A -85,B 0,C 180,E1 8636.071,E2 8636.071} C_VEL
LIN {X 0,Y 191.735,Z 581.359,A -85,B 0,C 180,E1 8630.697,E2 8630.697} C_VEL
LIN {X 0,Y 193.743,Z 585.979,A -85,B 0,C 180,E1 8626.572,E2 8626.572} C_VEL
LIN {X 0,Y 196.473,Z 592.191,A -85,B 0,C 180,E1 8621.915,E2 8621.915} C_VEL
LIN {X 0,Y 200.161,Z 601.977,A -85,B 0,C 180,E1 8616.133,E2 8616.133} C_VEL
LIN {X 0,Y 203.56,Z 612.083,A -85,B 0,C 180,E1 8611.226,E2 8611.226} C_VEL
LIN {X 0,Y 206.502,Z 621.523,A -85,B 0,C 180,E1 8607.408,E2 8607.408} C_VEL
LIN {X 0,Y 214.992,Z 637.224,A -85,B 0,C 180,E1 8604.456,E2 8604.456} C_VEL
LIN {X 0,Y 220.451,Z 648.705,A -85,B 0,C 180,E1 8602.685,E2 8602.685} C_VEL
LIN {X 0,Y 221,Z 665.514,A -85,B 0,C 180,E1 8601.849,E2 8601.849} C_VEL
LIN {X 0,Y 220.16,Z 679.055,A -85,B 0,C 180,E1 8601.462,E2 8601.462} C_VEL
LIN {X 0,Y 218.942,Z 686.719,A -85,B 0,C 180,E1 8601.401,E2 8601.401} C_VEL
LIN {X 0,Y 212.828,Z 706.999,A -85,B 0,C 180,E1 8601.87,E2 8601.87} C_VEL
LIN {X 0,Y 211.84,Z 713.583,A -85,B 0,C 180,E1 8601.808,E2 8601.808} C_VEL
LIN {X 0,Y 206.729,Z 797.578,A -85,B 0,C 180,E1 8599.255,E2 8599.255} C_VEL
LIN {X 0,Y 204.456,Z 815.858,A -85,B 0,C 180,E1 8598.265,E2 8598.265} C_VEL
LIN {X 0,Y 201.082,Z 833.54,A -85,B 0,C 180,E1 8596.861,E2 8596.861} C_VEL
LIN {X 0,Y 197.08,Z 849.92,A -85,B 0,C 180,E1 8595.049,E2 8595.049} C_VEL
LIN {X 0,Y 192.478,Z 865.801,A -85,B 0,C 180,E1 8592.68,E2 8592.68} C_VEL
LIN {X 0,Y 187.611,Z 880.763,A -85,B 0,C 180,E1 8589.758,E2 8589.758} C_VEL
LIN {X 0,Y 182.688,Z 894.734,A -85,B 0,C 180,E1 8586.235,E2 8586.235} C_VEL
LIN {X 0,Y 178.231,Z 907.186,A -85,B 0,C 180,E1 8582.206,E2 8582.206} C_VEL
LIN {X 0,Y 174.481,Z 918.135,A -85,B 0,C 180,E1 8577.658,E2 8577.658} C_VEL
LIN {X 0,Y 171.654,Z 927.63,A -85,B 0,C 180,E1 8572.611,E2 8572.611} C_VEL
LIN {X 0,Y 170.033,Z 935.651,A -85,B 0,C 180,E1 8567.101,E2 8567.101} C_VEL
LIN {X 0,Y 169.729,Z 941.754,A -85,B 0,C 180,E1 8561.557,E2 8561.557} C_VEL
LIN {X 0,Y 170.49,Z 946.08,A -85,B 0,C 180,E1 8556.063,E2 8556.063} C_VEL
LIN {X 0,Y 171.451,Z 948.409,A -85,B 0,C 180,E1 8551.341,E2 8551.341} C_VEL
LIN {X 0,Y 171.297,Z 949.093,A -85,B 0,C 180,E1 8548.332,E2 8548.332} C_VEL
LIN {X 0,Y 170.022,Z 948.935,A -85,B 0,C 180,E1 8543.25,E2 8543.25} C_VEL
LIN {X 0,Y 169.267,Z 947.004,A -85,B 0,C 180,E1 8537.034,E2 8537.034} C_VEL
LIN {X 0,Y 170.151,Z 943.3,A -85,B 0,C 180,E1 8530.794,E2 8530.794} C_VEL
LIN {X 0,Y 172.911,Z 937.779,A -85,B 0,C 180,E1 8524.672,E2 8524.672} C_VEL
LIN {X 0,Y 177.312,Z 930.751,A -85,B 0,C 180,E1 8519.134,E2 8519.134} C_VEL
LIN {X 0,Y 183.354,Z 921.696,A -85,B 0,C 180,E1 8513.926,E2 8513.926} C_VEL
LIN {X 0,Y 190.44,Z 911.078,A -85,B 0,C 180,E1 8509.39,E2 8509.39} C_VEL
LIN {X 0,Y 197.703,Z 899.778,A -85,B 0,C 180,E1 8505.75,E2 8505.75} C_VEL
LIN {X 0,Y 205.48,Z 886.6,A -85,B 0,C 180,E1 8502.517,E2 8502.517} C_VEL
LIN {X 0,Y 213.011,Z 872.238,A -85,B 0,C 180,E1 8499.885,E2 8499.885} C_VEL
LIN {X 0,Y 220.048,Z 856.805,A -85,B 0,C 180,E1 8497.768,E2 8497.768} C_VEL
LIN {X 0,Y 226.043,Z 841.241,A -85,B 0,C 180,E1 8496.183,E2 8496.183} C_VEL
LIN {X 0,Y 231.332,Z 824.181,A -85,B 0,C 180,E1 8494.914,E2 8494.914} C_VEL
LIN {X 0,Y 235.315,Z 806.341,A -85,B 0,C 180,E1 8493.985,E2 8493.985} C_VEL
LIN {X 0,Y 237.869,Z 787.727,A -85,B 0,C 180,E1 8493.332,E2 8493.332} C_VEL
LIN {X 0,Y 246.995,Z 677.548,A -85,B 0,C 180,E1 8490.486,E2 8490.486} C_VEL
LIN {X 0,Y 241.807,Z 667.782,A -85,B 0,C 180,E1 8487.321,E2 8487.321} C_VEL
LIN {X 0,Y 238.262,Z 661.845,A -85,B 0,C 180,E1 8484.878,E2 8484.878} C_VEL
LIN {X 0,Y 235.014,Z 656.605,A -85,B 0,C 180,E1 8482.249,E2 8482.249} C_VEL
LIN {X 0,Y 232.103,Z 652.263,A -85,B 0,C 180,E1 8479.503,E2 8479.503} C_VEL
LIN {X 0,Y 229.046,Z 648.082,A -85,B 0,C 180,E1 8475.832,E2 8475.832} C_VEL
LIN {X 0,Y 226.469,Z 644.623,A -85,B 0,C 180,E1 8471.201,E2 8471.201} C_VEL
LIN {X 0,Y 225.137,Z 643.653,A -85,B 0,C 180,E1 8465.351,E2 8465.351} C_VEL
LIN {X 0,Y 225.293,Z 644.234,A -85,B 0,C 180,E1 8462.543,E2 8462.543} C_VEL
LIN {X 0,Y 227.09,Z 647.576,A -85,B 0,C 180,E1 8456.845,E2 8456.845} C_VEL
LIN {X 0,Y 229.177,Z 651.598,A -85,B 0,C 180,E1 8453.36,E2 8453.36} C_VEL
LIN {X 0,Y 231.918,Z 656.364,A -85,B 0,C 180,E1 8450.069,E2 8450.069} C_VEL
LIN {X 0,Y 235.355,Z 662.834,A -85,B 0,C 180,E1 8446.8,E2 8446.8} C_VEL
LIN {X 0,Y 238.438,Z 669.05,A -85,B 0,C 180,E1 8444.307,E2 8444.307} C_VEL
LIN {X 0,Y 242.255,Z 677.318,A -85,B 0,C 180,E1 8441.625,E2 8441.625} C_VEL
LIN {X 0,Y 242.829,Z 679.233,A -85,B 0,C 180,E1 8441.204,E2 8441.204} C_VEL
LIN {X 0,Y 243.785,Z 697.531,A -85,B 0,C 180,E1 8439.499,E2 8439.499} C_VEL
LIN {X 0,Y 236.957,Z 773.639,A -85,B 0,C 180,E1 8437.387,E2 8437.387} C_VEL
LIN {X 0,Y 234.491,Z 790.098,A -85,B 0,C 180,E1 8436.568,E2 8436.568} C_VEL
LIN {X 0,Y 230.707,Z 806.698,A -85,B 0,C 180,E1 8435.354,E2 8435.354} C_VEL
LIN {X 0,Y 226.078,Z 821.633,A -85,B 0,C 180,E1 8433.852,E2 8433.852} C_VEL
LIN {X 0,Y 220.397,Z 836.085,A -85,B 0,C 180,E1 8431.914,E2 8431.914} C_VEL
LIN {X 0,Y 214.295,Z 848.913,A -85,B 0,C 180,E1 8429.66,E2 8429.66} C_VEL
LIN {X 0,Y 207.602,Z 860.72,A -85,B 0,C 180,E1 8426.918,E2 8426.918} C_VEL
LIN {X 0,Y 200.627,Z 871.396,A -85,B 0,C 180,E1 8423.625,E2 8423.625} C_VEL
LIN {X 0,Y 194.203,Z 879.935,A -85,B 0,C 180,E1 8420.085,E2 8420.085} C_VEL
LIN {X 0,Y 187.694,Z 887.497,A -85,B 0,C 180,E1 8415.745,E2 8415.745} C_VEL
LIN {X 0,Y 182.261,Z 893.024,A -85,B 0,C 180,E1 8411.161,E2 8411.161} C_VEL
LIN {X 0,Y 177.806,Z 896.782,A -85,B 0,C 180,E1 8406.18,E2 8406.18} C_VEL
LIN {X 0,Y 174.421,Z 898.898,A -85,B 0,C 180,E1 8400.669,E2 8400.669} C_VEL
LIN {X 0,Y 172.424,Z 899.114,A -85,B 0,C 180,E1 8395.226,E2 8395.226} C_VEL
LIN {X 0,Y 171.573,Z 897.484,A -85,B 0,C 180,E1 8389.395,E2 8389.395} C_VEL
LIN {X 0,Y 171.847,Z 894.331,A -85,B 0,C 180,E1 8384.139,E2 8384.139} C_VEL
LIN {X 0,Y 173.214,Z 889.078,A -85,B 0,C 180,E1 8378.627,E2 8378.627} C_VEL
LIN {X 0,Y 175.538,Z 882.285,A -85,B 0,C 180,E1 8373.588,E2 8373.588} C_VEL
LIN {X 0,Y 178.64,Z 873.956,A -85,B 0,C 180,E1 8369.034,E2 8369.034} C_VEL
LIN {X 0,Y 182.318,Z 864.261,A -85,B 0,C 180,E1 8364.963,E2 8364.963} C_VEL
LIN {X 0,Y 186.335,Z 853.099,A -85,B 0,C 180,E1 8361.356,E2 8361.356} C_VEL
LIN {X 0,Y 190.705,Z 839.841,A -85,B 0,C 180,E1 8358.045,E2 8358.045} C_VEL
LIN {X 0,Y 194.681,Z 826.04,A -85,B 0,C 180,E1 8355.422,E2 8355.422} C_VEL
LIN {X 0,Y 198.239,Z 811.352,A -85,B 0,C 180,E1 8353.29,E2 8353.29} C_VEL
LIN {X 0,Y 201.217,Z 795.689,A -85,B 0,C 180,E1 8351.605,E2 8351.605} C_VEL
LIN {X 0,Y 203.539,Z 778.311,A -85,B 0,C 180,E1 8350.306,E2 8350.306} C_VEL
LIN {X 0,Y 204.88,Z 760.485,A -85,B 0,C 180,E1 8349.501,E2 8349.501} C_VEL
LIN {X 0,Y 209.596,Z 685.605,A -85,B 0,C 180,E1 8347.089,E2 8347.089} C_VEL
LIN {X 0,Y 205.329,Z 643.21,A -85,B 0,C 180,E1 8343.986,E2 8343.986} C_VEL
LIN {X 0,Y 199.041,Z 630.245,A -85,B 0,C 180,E1 8341.534,E2 8341.534} C_VEL
LIN {X 0,Y 196.926,Z 625.685,A -85,B 0,C 180,E1 8340.494,E2 8340.494} C_VEL
LIN {X 0,Y 194.575,Z 615.177,A -85,B 0,C 180,E1 8335.579,E2 8335.579} C_VEL
LIN {X 0,Y 192.203,Z 606.429,A -85,B 0,C 180,E1 8330.816,E2 8330.816} C_VEL
LIN {X 0,Y 189.784,Z 598.539,A -85,B 0,C 180,E1 8325.768,E2 8325.768} C_VEL
LIN {X 0,Y 187.533,Z 592.089,A -85,B 0,C 180,E1 8320.791,E2 8320.791} C_VEL
LIN {X 0,Y 185.949,Z 588.106,A -85,B 0,C 180,E1 8317.031,E2 8317.031} C_VEL
LIN {X 0,Y 184.746,Z 584.906,A -85,B 0,C 180,E1 8313.545,E2 8313.545} C_VEL
LIN {X 0,Y 183.321,Z 581.335,A -85,B 0,C 180,E1 8308.684,E2 8308.684} C_VEL
LIN {X 0,Y 181.902,Z 577.645,A -85,B 0,C 180,E1 8300.865,E2 8300.865} C_VEL
LIN {X 0,Y 181.251,Z 576.815,A -85,B 0,C 180,E1 8294.701,E2 8294.701} C_VEL
LIN {X 0,Y 181.619,Z 577.21,A -85,B 0,C 180,E1 8288.23,E2 8288.23} C_VEL
LIN {X 0,Y 182.312,Z 578.345,A -85,B 0,C 180,E1 8284.089,E2 8284.089} C_VEL
LIN {X 0,Y 184.345,Z 582.595,A -85,B 0,C 180,E1 8276.269,E2 8276.269} C_VEL
LIN {X 0,Y 186.305,Z 587.237,A -85,B 0,C 180,E1 8270.919,E2 8270.919} C_VEL
LIN {X 0,Y 188.072,Z 591.352,A -85,B 0,C 180,E1 8267.098,E2 8267.098} C_VEL
LIN {X 0,Y 190.699,Z 597.597,A -85,B 0,C 180,E1 8262.296,E2 8262.296} C_VEL
LIN {X 0,Y 194.085,Z 606.904,A -85,B 0,C 180,E1 8256.63,E2 8256.63} C_VEL
LIN {X 0,Y 197.185,Z 616.419,A -85,B 0,C 180,E1 8251.864,E2 8251.864} C_VEL
LIN {X 0,Y 198.893,Z 621.736,A -85,B 0,C 180,E1 8249.613,E2 8249.613} C_VEL
LIN {X 0,Y 207.517,Z 637.329,A -85,B 0,C 180,E1 8246.352,E2 8246.352} C_VEL
LIN {X 0,Y 214.462,Z 651.665,A -85,B 0,C 180,E1 8243.933,E2 8243.933} C_VEL
LIN {X 0,Y 214.851,Z 666.295,A -85,B 0,C 180,E1 8243.189,E2 8243.189} C_VEL
LIN {X 0,Y 211.84,Z 713.583,A -85,B 0,C 180,E1 8241.808,E2 8241.808} C_VEL
LIN {X 0,Y 210.6,Z 721.248,A -85,B 0,C 180,E1 8241.755,E2 8241.755} C_VEL
LIN {X 0,Y 204.525,Z 741.533,A -85,B 0,C 180,E1 8242.254,E2 8242.254} C_VEL
LIN {X 0,Y 203.561,Z 748.117,A -85,B 0,C 180,E1 8242.187,E2 8242.187} C_VEL
LIN {X 0,Y 200.406,Z 797.178,A -85,B 0,C 180,E1 8240.638,E2 8240.638} C_VEL
LIN {X 0,Y 198.027,Z 815.516,A -85,B 0,C 180,E1 8239.621,E2 8239.621} C_VEL
LIN {X 0,Y 194.669,Z 832.51,A -85,B 0,C 180,E1 8238.248,E2 8238.248} C_VEL
LIN {X 0,Y 190.515,Z 848.937,A -85,B 0,C 180,E1 8236.407,E2 8236.407} C_VEL
LIN {X 0,Y 185.721,Z 864.853,A -85,B 0,C 180,E1 8233.987,E2 8233.987} C_VEL
LIN {X 0,Y 180.639,Z 879.819,A -85,B 0,C 180,E1 8230.99,E2 8230.99} C_VEL
LIN {X 0,Y 175.487,Z 893.788,A -85,B 0,C 180,E1 8227.359,E2 8227.359} C_VEL
LIN {X 0,Y 170.635,Z 906.655,A -85,B 0,C 180,E1 8223.023,E2 8223.023} C_VEL
LIN {X 0,Y 166.569,Z 917.927,A -85,B 0,C 180,E1 8218.069,E2 8218.069} C_VEL
LIN {X 0,Y 163.612,Z 927.486,A -85,B 0,C 180,E1 8212.647,E2 8212.647} C_VEL
LIN {X 0,Y 162.019,Z 935.315,A -85,B 0,C 180,E1 8206.864,E2 8206.864} C_VEL
LIN {X 0,Y 161.829,Z 941.464,A -85,B 0,C 180,E1 8200.774,E2 8200.774} C_VEL
LIN {X 0,Y 162.78,Z 945.536,A -85,B 0,C 180,E1 8194.937,E2 8194.937} C_VEL
LIN {X 0,Y 163.607,Z 947.334,A -85,B 0,C 180,E1 8190.705,E2 8190.705} C_VEL
LIN {X 0,Y 163.146,Z 947.925,A -85,B 0,C 180,E1 8187.384,E2 8187.384} C_VEL
LIN {X 0,Y 161.728,Z 947.477,A -85,B 0,C 180,E1 8181.472,E2 8181.472} C_VEL
LIN {X 0,Y 161.395,Z 945.246,A -85,B 0,C 180,E1 8174.924,E2 8174.924} C_VEL
LIN {X 0,Y 162.922,Z 941.238,A -85,B 0,C 180,E1 8168.401,E2 8168.401} C_VEL
LIN {X 0,Y 166.48,Z 935.332,A -85,B 0,C 180,E1 8162.073,E2 8162.073} C_VEL
LIN {X 0,Y 172.043,Z 927.425,A -85,B 0,C 180,E1 8156.096,E2 8156.096} C_VEL
LIN {X 0,Y 178.712,Z 918.272,A -85,B 0,C 180,E1 8151.048,E2 8151.048} C_VEL
LIN {X 0,Y 186.408,Z 907.477,A -85,B 0,C 180,E1 8146.651,E2 8146.651} C_VEL
LIN {X 0,Y 194.288,Z 895.617,A -85,B 0,C 180,E1 8143.06,E2 8143.06} C_VEL
LIN {X 0,Y 202.319,Z 882.271,A -85,B 0,C 180,E1 8140.015,E2 8140.015} C_VEL
LIN {X 0,Y 210.056,Z 867.763,A -85,B 0,C 180,E1 8137.537,E2 8137.537} C_VEL
LIN {X 0,Y 216.658,Z 853.408,A -85,B 0,C 180,E1 8135.699,E2 8135.699} C_VEL
LIN {X 0,Y 222.897,Z 837.126,A -85,B 0,C 180,E1 8134.158,E2 8134.158} C_VEL
LIN {X 0,Y 227.986,Z 820.228,A -85,B 0,C 180,E1 8133.005,E2 8133.005} C_VEL
LIN {X 0,Y 231.9,Z 802.102,A -85,B 0,C 180,E1 8132.131,E2 8132.131} C_VEL
LIN {X 0,Y 234.211,Z 783.988,A -85,B 0,C 180,E1 8131.546,E2 8131.546} C_VEL
LIN {X 0,Y 243.023,Z 681.778,A -85,B 0,C 180,E1 8128.922,E2 8128.922} C_VEL
LIN {X 0,Y 238.818,Z 673.652,A -85,B 0,C 180,E1 8126.145,E2 8126.145} C_VEL
LIN {X 0,Y 235.733,Z 668.261,A -85,B 0,C 180,E1 8123.828,E2 8123.828} C_VEL
LIN {X 0,Y 232.924,Z 663.622,A -85,B 0,C 180,E1 8121.399,E2 8121.399} C_VEL
LIN {X 0,Y 230.394,Z 659.694,A -85,B 0,C 180,E1 8118.863,E2 8118.863} C_VEL
LIN {X 0,Y 227.695,Z 655.784,A -85,B 0,C 180,E1 8115.406,E2 8115.406} C_VEL
LIN {X 0,Y 225.264,Z 652.425,A -85,B 0,C 180,E1 8110.744,E2 8110.744} C_VEL
LIN {X 0,Y 224.111,Z 651.597,A -85,B 0,C 180,E1 8105.119,E2 8105.119} C_VEL
LIN {X 0,Y 224.265,Z 652.226,A -85,B 0,C 180,E1 8102.555,E2 8102.555} C_VEL
LIN {X 0,Y 225.86,Z 655.353,A -85,B 0,C 180,E1 8097.208,E2 8097.208} C_VEL
LIN {X 0,Y 227.858,Z 659.422,A -85,B 0,C 180,E1 8093.701,E2 8093.701} C_VEL
LIN {X 0,Y 230.214,Z 663.792,A -85,B 0,C 180,E1 8090.689,E2 8090.689} C_VEL
LIN {X 0,Y 233.373,Z 670.049,A -85,B 0,C 180,E1 8087.504,E2 8087.504} C_VEL
LIN {X 0,Y 236.221,Z 676.179,A -85,B 0,C 180,E1 8085.036,E2 8085.036} C_VEL
